C07278=1030.289,161.461,393.307,169.169,44.738,158.424
C07279=1030.283,161.212,393.329,169.167,44.740,158.424
C07280=1030.277,160.963,393.352,169.164,44.742,158.424
C07281=1030.272,160.714,393.374,169.160,44.744,158.424
C07282=1030.266,160.465,393.396,169.158,44.746,158.425
C07283=1030.260,160.216,393.419,169.155,44.748,158.425
C07284=1030.255,159.967,393.442,169.152,44.749,158.425
C07285=1030.249,159.718,393.464,169.149,44.751,158.425
C07286=1030.243,159.469,393.486,169.145,44.754,158.425
C07287=1030.237,159.220,393.508,169.143,44.756,158.425
C07288=1030.231,158.971,393.531,169.141,44.758,158.425
C07289=1030.225,158.722,393.552,169.137,44.760,158.425
C07290=1030.218,158.473,393.575,169.134,44.762,158.425
C07291=1030.213,158.224,393.597,169.131,44.764,158.426
C07292=1030.207,157.975,393.618,169.128,44.766,158.426
C07293=1030.201,157.727,393.641,169.126,44.769,158.426
C07294=1030.195,157.477,393.663,169.122,44.771,158.426
C07295=1030.189,157.229,393.685,169.120,44.773,158.426
C07296=1030.183,156.980,393.707,169.116,44.775,158.426
C07297=1030.176,156.695,393.733,169.113,44.777,158.426
C07298=1030.170,156.411,393.757,169.110,44.780,158.427
C07299=1030.162,156.127,393.782,169.107,44.782,158.427
C07300=1030.156,155.842,393.807,169.103,44.785,158.427
C07301=1030.149,155.593,393.830,169.100,44.787,158.427
C07302=1030.144,155.344,393.851,169.097,44.789,158.427
C07303=1030.138,155.095,393.873,169.095,44.791,158.427
C07304=1030.132,154.846,393.895,169.091,44.794,158.428
C07305=1030.126,154.597,393.917,169.089,44.796,158.428
C07306=1030.120,154.348,393.939,169.086,44.798,158.428
C07307=1030.115,154.099,393.961,169.083,44.800,158.428
C07308=1030.108,153.851,393.983,169.080,44.802,158.428
C07309=1030.102,153.601,394.005,169.078,44.804,158.428
C07310=1030.096,153.352,394.026,169.074,44.807,158.429
C07311=1030.091,153.103,394.048,169.072,44.808,158.429
C07312=1030.085,152.855,394.070,169.068,44.811,158.429
C07313=1030.078,152.606,394.092,169.066,44.813,158.429
C07314=1030.072,152.356,394.114,169.063,44.815,158.429
C07315=1030.066,152.107,394.135,169.060,44.817,158.429
C07316=1030.060,151.859,394.157,169.057,44.819,158.429
C07317=1030.054,151.609,394.178,169.055,44.821,158.430
C07318=1030.049,151.360,394.201,169.051,44.823,158.430
C07319=1030.042,151.111,394.223,169.049,44.826,158.430
C07320=1030.037,150.863,394.244,169.046,44.828,158.430
C07321=1030.031,150.614,394.266,169.043,44.830,158.430
C07322=1030.025,150.364,394.287,169.040,44.832,158.430
C07323=1030.018,150.115,394.309,169.038,44.835,158.431
C07324=1030.013,149.867,394.330,169.034,44.837,158.431
C07325=1030.007,149.617,394.352,169.032,44.839,158.431
C07326=1030.000,149.368,394.373,169.029,44.841,158.431
C07327=1029.996,149.119,394.395,169.026,44.844,158.431
C07328=1029.989,148.870,394.417,169.023,44.846,158.431
C07329=1029.983,148.621,394.439,169.021,44.848,158.431
C07330=1029.977,148.373,394.461,169.017,44.850,158.431
C07331=1029.971,148.124,394.482,169.015,44.852,158.432
C07332=1029.965,147.875,394.504,169.012,44.854,158.432
C07333=1029.959,147.626,394.525,169.009,44.856,158.432
C07334=1029.953,147.377,394.547,169.006,44.858,158.432
C07335=1029.948,147.127,394.568,169.004,44.861,158.432
C07336=1029.941,146.878,394.589,169.000,44.863,158.433
C07337=1029.936,146.629,394.611,168.998,44.865,158.433
C07338=1029.930,146.380,394.632,168.995,44.867,158.433
C07339=1029.924,146.131,394.654,168.992,44.870,158.433
C07340=1029.918,145.883,394.675,168.989,44.872,158.433
C07341=1029.912,145.633,394.697,168.987,44.874,158.433
C07342=1029.905,145.384,394.718,168.983,44.877,158.434
C07343=1029.899,145.136,394.739,168.981,44.879,158.434
C07344=1029.893,144.887,394.761,168.978,44.881,158.434
C07345=1029.887,144.637,394.782,168.975,44.883,158.434
C07346=1029.882,144.388,394.803,168.972,44.885,158.434
C07347=1029.876,144.139,394.825,168.970,44.888,158.434
C07348=1029.869,143.890,394.846,168.967,44.890,158.435
C07349=1029.863,143.642,394.867,168.964,44.892,158.435
C07350=1029.857,143.392,394.888,168.962,44.895,158.435
C07351=1029.852,143.143,394.909,168.959,44.897,158.435
C07352=1029.846,142.894,394.931,168.955,44.899,158.435
C07353=1029.839,142.645,394.952,168.953,44.901,158.435
C07354=1029.834,142.397,394.974,168.951,44.903,158.436
C07355=1029.828,142.147,394.994,168.947,44.906,158.436
C07356=1029.822,141.899,395.015,168.945,44.908,158.436
C07357=1029.815,141.649,395.037,168.942,44.910,158.436
C07358=1029.809,141.400,395.058,168.940,44.912,158.436
C07359=1029.804,141.151,395.079,168.936,44.915,158.436
C07360=1029.798,140.902,395.101,168.934,44.917,158.437
C07361=1029.791,140.618,395.125,168.930,44.920,158.437
C07362=1029.784,140.333,395.149,168.928,44.922,158.437
C07363=1029.778,140.047,395.173,168.924,44.925,158.437
C07364=1029.771,139.763,395.197,168.921,44.927,158.437
C07365=1029.765,139.514,395.219,168.919,44.929,158.438
C07366=1029.759,139.265,395.239,168.916,44.931,158.438
C07367=1029.753,139.016,395.260,168.913,44.934,158.438
C07368=1029.747,138.768,395.282,168.910,44.936,158.438
C07369=1029.741,138.518,395.303,168.908,44.938,158.438
C07370=1029.735,138.269,395.323,168.905,44.941,158.438
C07371=1029.729,138.020,395.344,168.902,44.943,158.439
C07372=1029.723,137.770,395.366,168.899,44.946,158.439
C07373=1029.717,137.522,395.387,168.897,44.947,158.439
C07374=1029.711,137.272,395.407,168.893,44.950,158.439
C07375=1029.705,137.024,395.429,168.891,44.952,158.439
C07376=1029.699,136.774,395.449,168.888,44.954,158.439
C07377=1029.693,136.526,395.470,168.886,44.957,158.440
C07378=1029.687,136.276,395.491,168.883,44.959,158.440
C07379=1029.681,136.028,395.512,168.880,44.962,158.440
C07380=1029.675,135.778,395.533,168.878,44.964,158.440
C07381=1029.669,135.530,395.554,168.875,44.966,158.440
C07382=1029.663,135.280,395.574,168.872,44.968,158.441
C07383=1029.657,135.032,395.596,168.869,44.970,158.441
C07384=1029.651,134.782,395.616,168.867,44.973,158.441
C07385=1029.645,134.534,395.637,168.864,44.975,158.441
C07386=1029.638,134.284,395.658,168.861,44.978,158.441
C07387=1029.633,134.035,395.678,168.859,44.980,158.442
C07388=1029.627,133.786,395.700,168.856,44.982,158.442
C07389=1029.621,133.537,395.720,168.854,44.984,158.442
C07390=1029.615,133.288,395.741,168.850,44.987,158.442
C07391=1029.609,133.039,395.761,168.848,44.989,158.442
C07392=1029.603,132.789,395.782,168.845,44.991,158.442
C07393=1029.597,132.541,395.803,168.843,44.994,158.443
C07394=1029.591,132.292,395.824,168.839,44.996,158.443
C07395=1029.585,132.043,395.845,168.837,44.999,158.443
C07396=1029.579,131.794,395.865,168.834,45.001,158.443
C07397=1029.573,131.544,395.886,168.832,45.003,158.443
C07398=1029.567,131.296,395.907,168.830,45.005,158.444
C07399=1029.561,131.046,395.928,168.826,45.007,158.444
C07400=1029.555,130.797,395.948,168.824,45.010,158.444
C07401=1029.550,130.549,395.969,168.821,45.012,158.444
C07402=1029.543,130.299,395.989,168.819,45.015,158.444
C07403=1029.538,130.050,396.010,168.815,45.017,158.445
C07404=1029.531,129.800,396.030,168.813,45.019,158.445
C07405=1029.525,129.552,396.050,168.810,45.021,158.445
C07406=1029.518,129.303,396.071,168.808,45.024,158.445
C07407=1029.513,129.054,396.092,168.805,45.027,158.445
C07408=1029.507,128.804,396.112,168.802,45.029,158.446
C07409=1029.501,128.555,396.132,168.800,45.032,158.446
C07410=1029.494,128.306,396.152,168.797,45.033,158.446
C07411=1029.488,128.057,396.172,168.794,45.036,158.446
C07412=1029.482,127.808,396.193,168.792,45.038,158.446
C07413=1029.476,127.559,396.214,168.789,45.041,158.447
C07414=1029.470,127.310,396.234,168.787,45.044,158.447
C07415=1029.463,127.061,396.254,168.783,45.046,158.447
C07416=1029.458,126.811,396.275,168.781,45.048,158.447
C07417=1029.452,126.563,396.295,168.779,45.050,158.447
C07418=1029.445,126.313,396.315,168.776,45.053,158.448
C07419=1029.439,126.064,396.335,168.773,45.056,158.448
C07420=1029.434,125.814,396.356,168.770,45.058,158.448
C07421=1029.427,125.566,396.376,168.768,45.060,158.448
C07422=1029.421,125.317,396.396,168.766,45.062,158.448
C07423=1029.415,125.068,396.417,168.763,45.065,158.449
C07424=1029.409,124.819,396.437,168.760,45.067,158.449
C07425=1029.403,124.575,396.457,168.757,45.070,158.449
C07426=1029.397,124.332,396.476,168.755,45.072,158.449
C07427=1029.391,124.088,396.496,168.752,45.075,158.450
C07428=1029.386,123.845,396.516,168.750,45.077,158.450
C07429=1029.380,123.602,396.536,168.748,45.079,158.450
C07430=1029.374,123.358,396.555,168.744,45.081,158.450
C07431=1029.368,123.115,396.575,168.742,45.084,158.450
C07432=1029.362,122.871,396.595,168.739,45.086,158.450
C07433=1029.356,122.622,396.615,168.737,45.089,158.451
C07434=1029.350,122.373,396.635,168.734,45.091,158.451
C07435=1029.344,122.124,396.655,168.732,45.093,158.451
C07436=1029.337,121.875,396.675,168.728,45.095,158.451
C07437=1029.332,121.625,396.696,168.726,45.098,158.451
C07438=1029.326,121.377,396.716,168.724,45.101,158.452
C07439=1029.320,121.127,396.736,168.721,45.103,158.452
C07440=1029.314,120.878,396.756,168.719,45.105,158.452
C07441=1029.308,120.629,396.777,168.716,45.107,158.452
C07442=1029.302,120.380,396.797,168.713,45.110,158.453
C07443=1029.296,120.131,396.817,168.711,45.112,158.453
C07444=1029.290,119.882,396.837,168.708,45.115,158.453
C07445=1029.284,119.633,396.856,168.706,45.117,158.453
C07446=1029.279,119.383,396.877,168.703,45.119,158.453
C07447=1029.272,119.134,396.897,168.701,45.121,158.454
C07448=1029.266,118.885,396.917,168.698,45.124,158.454
C07449=1029.260,118.636,396.937,168.695,45.126,158.454
C07450=1029.254,118.388,396.957,168.693,45.129,158.454
C07451=1029.248,118.138,396.978,168.690,45.131,158.454
C07452=1029.242,117.889,396.998,168.688,45.134,158.455
C07453=1029.235,117.592,397.021,168.685,45.136,158.455
C07454=1029.229,117.296,397.045,168.681,45.139,158.455
C07455=1029.221,117.001,397.069,168.679,45.142,158.455
C07456=1029.214,116.704,397.093,168.676,45.145,158.456
C07457=1029.208,116.455,397.113,168.673,45.147,158.456
C07458=1029.202,116.206,397.133,168.671,45.149,158.456
C07459=1029.197,115.957,397.152,168.668,45.151,158.456
C07460=1029.190,115.707,397.172,168.665,45.154,158.456
C07461=1029.185,115.458,397.193,168.662,45.156,158.456
C07462=1029.179,115.209,397.213,168.660,45.159,158.457
C07463=1029.173,114.960,397.232,168.658,45.161,158.457
C07464=1029.167,114.711,397.252,168.655,45.164,158.457
C07465=1029.161,114.462,397.272,168.653,45.165,158.457
C07466=1029.155,114.213,397.292,168.650,45.167,158.457
C07467=1029.150,113.963,397.312,168.648,45.170,158.458
C07468=1029.144,113.714,397.332,168.644,45.172,158.458
C07469=1029.138,113.465,397.352,168.642,45.175,158.458
C07470=1029.132,113.217,397.372,168.639,45.177,158.458
C07471=1029.126,112.967,397.391,168.637,45.180,158.458
C07472=1029.119,112.718,397.412,168.635,45.182,158.459
C07473=1029.114,112.468,397.431,168.632,45.184,158.459
C07474=1029.108,112.219,397.451,168.630,45.187,158.459
C07475=1029.102,111.971,397.471,168.627,45.189,158.459
C07476=1029.096,111.721,397.490,168.624,45.192,158.459
C07477=1029.090,111.472,397.510,168.622,45.194,158.460
C07478=1029.084,111.222,397.530,168.619,45.196,158.460
C07479=1029.078,110.973,397.550,168.617,45.199,158.460
C07480=1029.072,110.724,397.569,168.614,45.201,158.460
C07481=1029.065,110.475,397.588,168.612,45.204,158.461
C07482=1029.059,110.227,397.608,168.610,45.206,158.461
C07483=1029.054,109.977,397.627,168.606,45.209,158.461
C07484=1029.048,109.728,397.647,168.604,45.211,158.461
C07485=1029.041,109.478,397.667,168.601,45.213,158.461
C07486=1029.035,109.229,397.686,168.599,45.216,158.462
C07487=1029.029,108.980,397.706,168.597,45.219,158.462
C07488=1029.023,108.731,397.725,168.594,45.220,158.462
C07489=1029.016,108.447,397.747,168.591,45.223,158.462
C07490=1029.009,108.162,397.769,168.588,45.227,158.463
C07491=1029.002,107.877,397.791,168.586,45.230,158.463
C07492=1028.995,107.591,397.814,168.582,45.232,158.463
C07493=1028.989,107.342,397.834,168.580,45.234,158.463
C07494=1028.983,107.093,397.853,168.577,45.237,158.463
C07495=1028.977,106.844,397.872,168.575,45.240,158.464
C07496=1028.971,106.595,397.892,168.573,45.242,158.464
C07497=1028.965,106.345,397.911,168.569,45.245,158.464
C07498=1028.959,106.096,397.929,168.567,45.247,158.464
C07499=1028.953,105.847,397.949,168.564,45.249,158.464
C07500=1028.947,105.598,397.969,168.562,45.252,158.465
C07501=1028.941,105.349,397.989,168.560,45.254,158.465
C07502=1028.935,105.100,398.007,168.557,45.257,158.465
C07503=1028.929,104.851,398.027,168.555,45.259,158.465
C07504=1028.922,104.601,398.047,168.553,45.261,158.466
C07505=1028.916,104.352,398.065,168.549,45.264,158.466
C07506=1028.910,104.102,398.085,168.547,45.267,158.466
C07507=1028.905,103.853,398.104,168.544,45.269,158.466
C07508=1028.899,103.604,398.124,168.542,45.271,158.466
C07509=1028.892,103.355,398.143,168.540,45.273,158.467
C07510=1028.886,103.106,398.162,168.537,45.276,158.467
C07511=1028.880,102.857,398.182,168.535,45.279,158.467
C07512=1028.874,102.608,398.200,168.532,45.281,158.467
C07513=1028.868,102.358,398.220,168.530,45.283,158.468
C07514=1028.863,102.109,398.239,168.527,45.286,158.468
C07515=1028.857,101.860,398.259,168.524,45.288,158.468
C07516=1028.850,101.611,398.278,168.522,45.291,158.468
C07517=1028.845,101.362,398.297,168.519,45.293,158.468
C07518=1028.839,101.112,398.316,168.517,45.296,158.469
C07519=1028.832,100.864,398.335,168.515,45.298,158.469
C07520=1028.826,100.614,398.355,168.512,45.300,158.469
C07521=1028.821,100.365,398.374,168.510,45.303,158.469
C07522=1028.815,100.115,398.393,168.507,45.305,158.469
C07523=1028.809,99.866,398.412,168.505,45.308,158.470
C07524=1028.803,99.617,398.431,168.502,45.310,158.470
C07525=1028.796,99.368,398.450,168.499,45.312,158.470
C07526=1028.791,99.119,398.470,168.497,45.315,158.470
C07527=1028.784,98.870,398.488,168.495,45.318,158.471
C07528=1028.778,98.621,398.507,168.492,45.320,158.471
C07529=1028.772,98.371,398.526,168.490,45.322,158.471
C07530=1028.766,98.122,398.545,168.488,45.325,158.471
C07531=1028.760,97.873,398.564,168.484,45.328,158.471
C07532=1028.753,97.623,398.583,168.482,45.330,158.472
C07533=1028.748,97.374,398.602,168.479,45.333,158.472
C07534=1028.741,97.125,398.621,168.477,45.335,158.472
C07535=1028.735,96.876,398.639,168.475,45.337,158.472
C07536=1028.729,96.626,398.658,168.472,45.340,158.473
C07537=1028.723,96.378,398.677,168.470,45.343,158.473
C07538=1028.718,96.128,398.696,168.468,45.345,158.473
C07539=1028.711,95.879,398.715,168.464,45.348,158.473
C07540=1028.705,95.630,398.733,168.462,45.350,158.473
C07541=1028.699,95.381,398.753,168.460,45.353,158.474
C07542=1028.693,95.132,398.771,168.457,45.355,158.474
C07543=1028.687,94.882,398.790,168.455,45.358,158.474
C07544=1028.681,94.633,398.809,168.452,45.360,158.474
C07545=1028.675,94.384,398.828,168.450,45.362,158.474
C07546=1028.669,94.135,398.847,168.448,45.365,158.475
C07547=1028.662,93.885,398.866,168.445,45.368,158.475
C07548=1028.656,93.636,398.885,168.443,45.370,158.475
C07549=1028.651,93.388,398.903,168.439,45.373,158.475
C07550=1028.645,93.138,398.922,168.437,45.375,158.476
C07551=1028.638,92.889,398.941,168.435,45.377,158.476
C07552=1028.632,92.639,398.959,168.432,45.380,158.476
C07553=1028.626,92.354,398.981,168.430,45.383,158.476
C07554=1028.619,92.069,399.003,168.427,45.385,158.477
C07555=1028.611,91.784,399.024,168.424,45.388,158.477
C07556=1028.605,91.500,399.045,168.421,45.391,158.477
C07557=1028.599,91.251,399.064,168.419,45.394,158.477
C07558=1028.593,91.001,399.083,168.416,45.396,158.477
C07559=1028.587,90.752,399.102,168.414,45.398,158.478
C07560=1028.581,90.502,399.120,168.412,45.401,158.478
C07561=1028.575,90.253,399.139,168.409,45.403,158.478
C07562=1028.568,90.004,399.158,168.407,45.406,158.478
C07563=1028.563,89.755,399.176,168.405,45.408,158.479
C07564=1028.557,89.506,399.195,168.401,45.411,158.479
C07565=1028.551,89.256,399.213,168.399,45.413,158.479
C07566=1028.544,89.007,399.232,168.397,45.416,158.479
C07567=1028.538,88.758,399.250,168.394,45.419,158.480
C07568=1028.533,88.508,399.269,168.392,45.421,158.480
C07569=1028.526,88.259,399.288,168.389,45.423,158.480
C07570=1028.520,88.010,399.306,168.387,45.426,158.480
C07571=1028.514,87.761,399.324,168.385,45.429,158.480
C07572=1028.508,87.511,399.342,168.381,45.431,158.481
C07573=1028.501,87.262,399.361,168.379,45.434,158.481
C07574=1028.495,87.013,399.379,168.377,45.436,158.481
C07575=1028.489,86.763,399.398,168.374,45.439,158.481
C07576=1028.483,86.515,399.416,168.372,45.442,158.482
C07577=1028.478,86.265,399.434,168.370,45.444,158.482
C07578=1028.471,86.016,399.453,168.367,45.446,158.482
C07579=1028.465,85.767,399.472,168.365,45.449,158.482
C07580=1028.459,85.517,399.490,168.363,45.452,158.483
C07581=1028.453,85.269,399.508,168.359,45.454,158.483
C07582=1028.446,85.019,399.527,168.357,45.457,158.483
C07583=1028.440,84.770,399.545,168.355,45.459,158.483
C07584=1028.434,84.521,399.563,168.352,45.461,158.483
C07585=1028.428,84.271,399.581,168.350,45.464,158.484
C07586=1028.422,84.022,399.599,168.347,45.467,158.484
C07587=1028.416,83.773,399.617,168.345,45.469,158.484
C07588=1028.410,83.523,399.637,168.343,45.471,158.484
C07589=1028.404,83.274,399.655,168.340,45.474,158.484
C07590=1028.398,83.025,399.673,168.338,45.477,158.485
C07591=1028.392,82.776,399.691,168.335,45.479,158.485
C07592=1028.386,82.526,399.709,168.332,45.482,158.485
C07593=1028.379,82.277,399.728,168.330,45.484,158.485
C07594=1028.374,82.028,399.746,168.328,45.487,158.486
C07595=1028.367,81.779,399.764,168.325,45.489,158.486
C07596=1028.361,81.529,399.782,168.323,45.492,158.486
C07597=1028.355,81.280,399.801,168.321,45.494,158.486
C07598=1028.349,81.031,399.818,168.318,45.496,158.486
C07599=1028.343,80.782,399.837,168.316,45.499,158.487
C07600=1028.337,80.532,399.856,168.313,45.502,158.487
C07601=1028.331,80.283,399.874,168.311,45.504,158.487
C07602=1028.325,80.034,399.892,168.309,45.506,158.487
C07603=1028.319,79.785,399.910,168.306,45.509,158.488
C07604=1028.313,79.535,399.928,168.303,45.511,158.488
C07605=1028.307,79.286,399.947,168.301,45.514,158.488
C07606=1028.301,79.037,399.965,168.298,45.517,158.488
C07607=1028.295,78.787,399.982,168.296,45.519,158.488
C07608=1028.289,78.539,400.001,168.293,45.521,158.489
C07609=1028.283,78.289,400.019,168.291,45.524,158.489
C07610=1028.276,78.040,400.037,168.289,45.526,158.489
C07611=1028.271,77.791,400.055,168.286,45.529,158.489
C07612=1028.265,77.541,400.073,168.284,45.532,158.490
C07613=1028.258,77.292,400.091,168.281,45.534,158.490
C07614=1028.253,77.043,400.109,168.279,45.536,158.490
C07615=1028.247,76.793,400.127,168.277,45.539,158.490
C07616=1028.240,76.544,400.146,168.275,45.542,158.490
C07617=1028.234,76.259,400.166,168.271,45.545,158.491
C07618=1028.226,75.974,400.187,168.268,45.547,158.491
C07619=1028.219,75.689,400.207,168.266,45.550,158.491
C07620=1028.213,75.403,400.227,168.262,45.553,158.491
C07621=1028.206,75.154,400.246,168.260,45.556,158.492
C07622=1028.199,74.905,400.263,168.258,45.558,158.492
C07623=1028.194,74.656,400.280,168.256,45.561,158.492
C07624=1028.188,74.406,400.298,168.253,45.563,158.492
C07625=1028.182,74.158,400.317,168.251,45.566,158.493
C07626=1028.176,73.908,400.335,168.249,45.569,158.493
C07627=1028.169,73.659,400.352,168.246,45.571,158.493
C07628=1028.163,73.409,400.369,168.244,45.573,158.493
C07629=1028.157,73.160,400.387,168.240,45.576,158.493
C07630=1028.151,72.911,400.406,168.238,45.579,158.494
C07631=1028.145,72.662,400.424,168.236,45.581,158.494
C07632=1028.139,72.412,400.441,168.233,45.584,158.494
C07633=1028.133,72.163,400.459,168.231,45.586,158.494
C07634=1028.127,71.913,400.476,168.229,45.589,158.495
C07635=1028.120,71.664,400.495,168.226,45.591,158.495
C07636=1028.115,71.415,400.513,168.224,45.594,158.495
C07637=1028.108,71.166,400.530,168.222,45.596,158.495
C07638=1028.103,70.917,400.548,168.219,45.599,158.496
C07639=1028.096,70.667,400.566,168.217,45.601,158.496
C07640=1028.090,70.418,400.583,168.215,45.604,158.496
C07641=1028.084,70.169,400.600,168.211,45.607,158.496
C07642=1028.078,69.919,400.618,168.209,45.609,158.496
C07643=1028.072,69.670,400.636,168.206,45.611,158.496
C07644=1028.065,69.421,400.654,168.204,45.614,158.497
C07645=1028.060,69.172,400.672,168.202,45.617,158.497
C07646=1028.054,68.922,400.689,168.199,45.619,158.497
C07647=1028.047,68.672,400.707,168.197,45.622,158.497
C07648=1028.041,68.424,400.724,168.195,45.624,158.498
C07649=1028.035,68.174,400.742,168.193,45.627,158.498
C07650=1028.029,67.925,400.759,168.190,45.629,158.498
C07651=1028.023,67.675,400.777,168.188,45.632,158.498
C07652=1028.017,67.426,400.795,168.184,45.635,158.499
C07653=1028.010,67.177,400.812,168.182,45.637,158.499
C07654=1028.005,66.928,400.830,168.180,45.639,158.499
C07655=1027.999,66.678,400.848,168.177,45.642,158.499
C07656=1027.992,66.429,400.865,168.175,45.645,158.499
C07657=1027.986,66.180,400.883,168.173,45.647,158.500
C07658=1027.979,65.930,400.900,168.170,45.649,158.500
C07659=1027.974,65.681,400.917,168.168,45.652,158.500
C07660=1027.967,65.431,400.934,168.166,45.655,158.500
C07661=1027.962,65.182,400.952,168.163,45.658,158.501
C07662=1027.955,64.933,400.969,168.160,45.660,158.501
C07663=1027.950,64.684,400.987,168.158,45.663,158.501
C07664=1027.943,64.434,401.004,168.155,45.665,158.501
C07665=1027.937,64.185,401.021,168.153,45.668,158.501
C07666=1027.931,63.935,401.039,168.150,45.670,158.502
C07667=1027.925,63.687,401.056,168.148,45.673,158.502
C07668=1027.919,63.437,401.074,168.146,45.675,158.502
C07669=1027.913,63.188,401.091,168.144,45.678,158.502
C07670=1027.906,62.938,401.108,168.141,45.681,158.503
C07671=1027.900,62.689,401.125,168.138,45.684,158.503
C07672=1027.893,62.440,401.143,168.136,45.686,158.503
C07673=1027.887,62.190,401.159,168.133,45.688,158.503
C07674=1027.881,61.941,401.176,168.131,45.691,158.504
C07675=1027.875,61.692,401.194,168.129,45.694,158.504
C07676=1027.869,61.442,401.211,168.126,45.697,158.504
C07677=1027.862,61.193,401.228,168.124,45.699,158.504
C07678=1027.856,60.943,401.245,168.121,45.702,158.505
C07679=1027.850,60.695,401.262,168.119,45.705,158.505
C07680=1027.843,60.445,401.279,168.116,45.708,158.505
C07681=1027.836,60.160,401.298,168.113,45.711,158.505
C07682=1027.829,59.874,401.319,168.111,45.713,158.506
C07683=1027.822,59.590,401.338,168.107,45.716,158.506
C07684=1027.816,59.304,401.357,168.105,45.720,158.506
C07685=1027.809,59.055,401.375,168.103,45.722,158.506
C07686=1027.803,58.806,401.391,168.100,45.725,158.506
C07687=1027.796,58.556,401.408,168.097,45.727,158.507
C07688=1027.790,58.307,401.426,168.095,45.730,158.507
C07689=1027.784,58.057,401.442,168.093,45.733,158.507
C07690=1027.778,57.808,401.459,168.091,45.735,158.508
C07691=1027.772,57.559,401.476,168.088,45.738,158.508
C07692=1027.765,57.309,401.494,168.086,45.740,158.508
C07693=1027.759,57.060,401.511,168.082,45.743,158.508
C07694=1027.753,56.810,401.527,168.080,45.746,158.508
C07695=1027.746,56.562,401.544,168.078,45.748,158.509
C07696=1027.740,56.312,401.561,168.076,45.751,158.509
C07697=1027.734,56.063,401.578,168.073,45.754,158.509
C07698=1027.728,55.814,401.595,168.071,45.756,158.509
C07699=1027.722,55.564,401.612,168.069,45.759,158.510
C07700=1027.715,55.315,401.629,168.066,45.761,158.510
C07701=1027.710,55.065,401.646,168.063,45.764,158.510
C07702=1027.703,54.816,401.663,168.061,45.767,158.510
C07703=1027.697,54.567,401.679,168.058,45.769,158.510
C07704=1027.690,54.317,401.697,168.056,45.772,158.511
C07705=1027.685,54.068,401.714,168.054,45.774,158.511
C07706=1027.679,53.819,401.730,168.051,45.777,158.511
C07707=1027.672,53.569,401.747,168.049,45.780,158.511
C07708=1027.666,53.320,401.764,168.047,45.782,158.512
C07709=1027.661,53.070,401.781,168.043,45.785,158.512
C07710=1027.654,52.821,401.798,168.041,45.788,158.512
C07711=1027.648,52.572,401.815,168.039,45.790,158.512
C07712=1027.642,52.323,401.832,168.036,45.792,158.512
C07713=1027.635,52.073,401.848,168.034,45.795,158.513
C07714=1027.630,51.824,401.866,168.032,45.798,158.513
C07715=1027.624,51.574,401.882,168.029,45.801,158.513
C07716=1027.617,51.325,401.899,168.027,45.803,158.513
C07717=1027.611,51.076,401.916,168.025,45.805,158.514
C07718=1027.605,50.827,401.933,168.021,45.808,158.514
C07719=1027.599,50.577,401.950,168.019,45.811,158.514
C07720=1027.593,50.327,401.966,168.016,45.813,158.514
C07721=1027.587,50.079,401.983,168.014,45.816,158.514
C07722=1027.581,49.829,401.999,168.012,45.818,158.515
C07723=1027.575,49.579,402.017,168.009,45.820,158.515
C07724=1027.569,49.330,402.033,168.007,45.823,158.515
C07725=1027.563,49.081,402.050,168.005,45.826,158.515
C07726=1027.556,48.832,402.067,168.003,45.829,158.516
C07727=1027.550,48.582,402.083,168.000,45.831,158.516
C07728=1027.544,48.333,402.101,167.997,45.834,158.516
C07729=1027.538,48.084,402.117,167.994,45.836,158.516
C07730=1027.532,47.834,402.134,167.992,45.838,158.516
C07731=1027.526,47.585,402.151,167.990,45.841,158.516
C07732=1027.520,47.335,402.167,167.987,45.844,158.517
C07733=1027.514,47.086,402.184,167.985,45.846,158.517
C07734=1027.508,46.837,402.201,167.983,45.849,158.517
C07735=1027.502,46.587,402.217,167.980,45.851,158.517
C07736=1027.496,46.338,402.234,167.978,45.853,158.517
C07737=1027.489,46.089,402.251,167.976,45.856,158.518
C07738=1027.484,45.839,402.267,167.973,45.859,158.518
C07739=1027.478,45.589,402.284,167.971,45.861,158.518
C07740=1027.472,45.340,402.300,167.967,45.864,158.518
C07741=1027.466,45.091,402.317,167.965,45.866,158.519
C07742=1027.460,44.842,402.334,167.963,45.869,158.519
C07743=1027.454,44.592,402.350,167.960,45.871,158.519
C07744=1027.448,44.343,402.367,167.958,45.873,158.519
C07745=1027.441,44.057,402.386,167.956,45.876,158.519
C07746=1027.434,43.772,402.406,167.952,45.879,158.519
C07747=1027.428,43.486,402.424,167.950,45.882,158.520
C07748=1027.420,43.201,402.443,167.947,45.885,158.520
C07749=1027.415,42.951,402.460,167.944,45.887,158.520
C07750=1027.409,42.702,402.476,167.942,45.890,158.520
C07751=1027.403,42.452,402.493,167.940,45.893,158.521
C07752=1027.396,42.203,402.508,167.937,45.895,158.521
C07753=1027.389,41.953,402.525,167.934,45.898,158.521
C07754=1027.383,41.705,402.542,167.932,45.901,158.521
C07755=1027.377,41.455,402.558,167.930,45.903,158.522
C07756=1027.371,41.206,402.574,167.927,45.905,158.522
C07757=1027.365,40.957,402.591,167.925,45.908,158.522
C07758=1027.359,40.707,402.607,167.923,45.911,158.522
C07759=1027.353,40.457,402.624,167.920,45.914,158.522
C07760=1027.347,40.208,402.640,167.918,45.916,158.523
C07761=1027.341,39.958,402.656,167.914,45.919,158.523
C07762=1027.335,39.709,402.672,167.912,45.921,158.523
C07763=1027.328,39.460,402.688,167.910,45.924,158.523
C07764=1027.322,39.211,402.704,167.907,45.926,158.523
C07765=1027.316,38.961,402.720,167.905,45.929,158.524
C07766=1027.310,38.711,402.737,167.903,45.931,158.524
C07767=1027.304,38.462,402.753,167.901,45.934,158.524
C07768=1027.298,38.213,402.770,167.898,45.936,158.524
C07769=1027.292,37.963,402.786,167.895,45.939,158.524
C07770=1027.286,37.714,402.802,167.893,45.942,158.525
C07771=1027.280,37.465,402.818,167.890,45.944,158.525
C07772=1027.274,37.215,402.835,167.888,45.947,158.525
C07773=1027.268,36.966,402.851,167.885,45.949,158.525
C07774=1027.261,36.716,402.867,167.883,45.952,158.526
C07775=1027.255,36.467,402.883,167.881,45.954,158.526
C07776=1027.249,36.217,402.899,167.877,45.957,158.526
C07777=1027.242,35.968,402.915,167.875,45.960,158.526
C07778=1027.237,35.718,402.931,167.873,45.963,158.526
C07779=1027.231,35.469,402.947,167.871,45.965,158.527
C07780=1027.224,35.220,402.963,167.868,45.968,158.527
C07781=1027.218,34.971,402.979,167.865,45.970,158.527
C07782=1027.212,34.721,402.995,167.862,45.973,158.527
C07783=1027.205,34.472,403.011,167.860,45.976,158.527
C07784=1027.200,34.222,403.026,167.858,45.979,158.528
C07785=1027.193,33.972,403.043,167.856,45.981,158.528
C07786=1027.187,33.723,403.059,167.853,45.983,158.528
C07787=1027.181,33.474,403.075,167.850,45.986,158.528
C07788=1027.175,33.225,403.091,167.848,45.989,158.528
C07789=1027.168,32.975,403.106,167.845,45.992,158.529
C07790=1027.162,32.726,403.122,167.843,45.995,158.529
C07791=1027.156,32.476,403.139,167.841,45.997,158.529
C07792=1027.150,32.227,403.154,167.838,45.999,158.529
C07793=1027.144,31.978,403.170,167.835,46.002,158.530
C07794=1027.138,31.728,403.186,167.833,46.005,158.530
C07795=1027.131,31.479,403.202,167.830,46.007,158.530
C07796=1027.125,31.230,403.218,167.828,46.010,158.530
C07797=1027.119,30.980,403.234,167.826,46.013,158.530
C07798=1027.113,30.730,403.249,167.823,46.015,158.531
C07799=1027.107,30.481,403.265,167.820,46.018,158.531
C07800=1027.100,30.232,403.281,167.818,46.020,158.531
C07801=1027.095,29.982,403.297,167.815,46.023,158.531
C07802=1027.089,29.733,403.313,167.813,46.026,158.531
C07803=1027.082,29.484,403.328,167.811,46.028,158.532
C07804=1027.077,29.234,403.344,167.808,46.031,158.532
C07805=1027.071,28.984,403.360,167.805,46.034,158.532
C07806=1027.064,28.735,403.376,167.803,46.036,158.532
C07807=1027.058,28.485,403.391,167.800,46.038,158.532
C07808=1027.052,28.236,403.408,167.798,46.041,158.533
C07809=1027.045,27.951,403.425,167.795,46.044,158.533
C07810=1027.038,27.665,403.444,167.792,46.047,158.533
C07811=1027.031,27.380,403.462,167.789,46.050,158.533
C07812=1027.024,27.094,403.479,167.786,46.054,158.534
C07813=1027.018,26.845,403.495,167.784,46.056,158.534
C07814=1027.011,26.596,403.511,167.781,46.058,158.534
C07815=1027.005,26.346,403.526,167.779,46.061,158.534
C07816=1026.999,26.097,403.542,167.777,46.064,158.534
C07817=1026.993,25.847,403.557,167.774,46.067,158.535
C07818=1026.987,25.598,403.573,167.771,46.069,158.535
C07819=1026.980,25.348,403.588,167.769,46.072,158.535
C07820=1026.974,25.099,403.604,167.767,46.074,158.535
C07821=1026.968,24.849,403.619,167.764,46.077,158.536
C07822=1026.961,24.600,403.635,167.761,46.080,158.536
C07823=1026.956,24.350,403.651,167.759,46.083,158.536
C07824=1026.949,24.101,403.666,167.756,46.085,158.536
C07825=1026.944,23.852,403.681,167.754,46.088,158.536
C07826=1026.937,23.602,403.696,167.752,46.090,158.537
C07827=1026.932,23.353,403.713,167.748,46.093,158.537
C07828=1026.925,23.103,403.728,167.746,46.096,158.537
C07829=1026.918,22.854,403.743,167.744,46.098,158.537
C07830=1026.913,22.604,403.759,167.741,46.101,158.537
C07831=1026.906,22.355,403.774,167.739,46.104,158.538
C07832=1026.900,22.105,403.790,167.736,46.107,158.538
C07833=1026.894,21.855,403.805,167.733,46.109,158.538
C07834=1026.888,21.607,403.820,167.731,46.111,158.538
C07835=1026.882,21.357,403.836,167.729,46.114,158.538
C07836=1026.876,21.108,403.851,167.727,46.117,158.539
C07837=1026.869,20.858,403.866,167.723,46.119,158.539
C07838=1026.864,20.608,403.882,167.721,46.122,158.539
C07839=1026.857,20.359,403.898,167.718,46.125,158.539
C07840=1026.851,20.109,403.913,167.716,46.128,158.539
C07841=1026.845,19.860,403.928,167.714,46.130,158.540
C07842=1026.839,19.611,403.943,167.710,46.133,158.540
C07843=1026.833,19.361,403.959,167.708,46.135,158.540
C07844=1026.827,19.112,403.974,167.706,46.138,158.540
C07845=1026.820,18.863,403.990,167.703,46.140,158.540
C07846=1026.814,18.613,404.005,167.700,46.143,158.541
C07847=1026.808,18.363,404.020,167.698,46.146,158.541
C07848=1026.802,18.114,404.035,167.696,46.149,158.541
C07849=1026.796,17.865,404.050,167.693,46.151,158.541
C07850=1026.790,17.615,404.066,167.691,46.153,158.541
C07851=1026.784,17.365,404.081,167.688,46.156,158.542
C07852=1026.777,17.116,404.096,167.685,46.159,158.542
C07853=1026.771,16.866,404.111,167.683,46.162,158.542
C07854=1026.765,16.618,404.126,167.681,46.165,158.542
C07855=1026.759,16.368,404.141,167.677,46.167,158.542
C07856=1026.753,16.118,404.156,167.675,46.170,158.543
C07857=1026.746,15.868,404.171,167.673,46.172,158.543
C07858=1026.740,15.619,404.186,167.670,46.175,158.543
C07859=1026.735,15.370,404.202,167.668,46.177,158.543
C07860=1026.728,15.121,404.217,167.665,46.180,158.543
C07861=1026.722,14.871,404.232,167.662,46.183,158.544
C07862=1026.715,14.621,404.247,167.660,46.186,158.544
C07863=1026.710,14.372,404.262,167.658,46.188,158.544
C07864=1026.704,14.122,404.277,167.654,46.191,158.544
C07865=1026.698,13.873,404.292,167.652,46.194,158.544
C07866=1026.691,13.624,404.308,167.650,46.196,158.545
C07867=1026.685,13.375,404.322,167.648,46.199,158.545
C07868=1026.679,13.125,404.337,167.644,46.201,158.545
C07869=1026.672,12.875,404.352,167.642,46.204,158.545
C07870=1026.666,12.626,404.367,167.640,46.207,158.545
C07871=1026.660,12.376,404.382,167.636,46.210,158.546
C07872=1026.654,12.127,404.397,167.634,46.213,158.546
C07873=1026.647,11.843,404.414,167.631,46.216,158.546
C07874=1026.639,11.558,404.431,167.629,46.219,158.546
C07875=1026.633,11.274,404.447,167.625,46.222,158.547
C07876=1026.626,10.990,404.464,167.622,46.225,158.547
C07877=1026.619,10.740,404.479,167.620,46.228,158.547
C07878=1026.613,10.490,404.494,167.618,46.231,158.547
C07879=1026.607,10.241,404.508,167.614,46.234,158.548
C07880=1026.601,9.992,404.523,167.612,46.236,158.548
C07881=1026.594,9.742,404.538,167.610,46.238,158.548
C07882=1026.588,9.493,404.553,167.606,46.241,158.548
C07883=1026.582,9.244,404.568,167.604,46.244,158.548
C07884=1026.576,8.994,404.583,167.602,46.247,158.549
C07885=1026.569,8.744,404.597,167.600,46.250,158.549
C07886=1026.563,8.495,404.612,167.596,46.253,158.549
C07887=1026.557,8.246,404.627,167.594,46.255,158.549
C07888=1026.550,7.996,404.641,167.592,46.258,158.549
C07889=1026.545,7.747,404.655,167.588,46.261,158.549
C07890=1026.538,7.497,404.670,167.586,46.263,158.550
C07891=1026.532,7.247,404.685,167.584,46.266,158.550
C07892=1026.526,6.998,404.700,167.582,46.269,158.550
C07893=1026.520,6.749,404.715,167.578,46.271,158.550
C07894=1026.513,6.498,404.729,167.576,46.274,158.551
C07895=1026.508,6.250,404.743,167.573,46.277,158.551
C07896=1026.501,6.000,404.758,167.570,46.280,158.551
C07897=1026.496,5.751,404.773,167.568,46.283,158.551
C07898=1026.489,5.501,404.788,167.565,46.285,158.551
C07899=1026.483,5.252,404.803,167.563,46.287,158.552
C07900=1026.477,5.002,404.817,167.560,46.290,158.552
C07901=1026.471,4.752,404.832,167.558,46.293,158.552
C07902=1026.465,4.503,404.847,167.555,46.295,158.552
C07903=1026.459,4.254,404.861,167.552,46.298,158.552
C07904=1026.452,4.004,404.875,167.550,46.301,158.552
C07905=1026.446,3.755,404.889,167.547,46.304,158.553
C07906=1026.440,3.505,404.904,167.545,46.307,158.553
C07907=1026.434,3.256,404.919,167.542,46.309,158.553
C07908=1026.428,3.006,404.933,167.539,46.312,158.553
C07909=1026.422,2.756,404.948,167.537,46.314,158.553
C07910=1026.416,2.507,404.963,167.534,46.317,158.554
C07911=1026.409,2.258,404.978,167.531,46.319,158.554
C07912=1026.404,2.008,404.991,167.529,46.322,158.554
C07913=1026.398,1.758,405.006,167.527,46.325,158.554
C07914=1026.392,1.510,405.021,167.523,46.327,158.554
C07915=1026.386,1.259,405.035,167.521,46.330,158.554
C07916=1026.379,1.010,405.050,167.519,46.333,158.555
C07917=1026.373,0.761,405.064,167.515,46.336,158.555
C07918=1026.367,0.511,405.078,167.513,46.338,158.555
C07919=1026.361,0.262,405.093,167.511,46.341,158.555
C07920=1026.355,0.012,405.108,167.508,46.343,158.556
C07921=1026.349,-0.238,405.122,167.505,46.346,158.556
C07922=1026.343,-0.487,405.137,167.503,46.349,158.556
C07923=1026.337,-0.736,405.151,167.500,46.351,158.556
C07924=1026.331,-0.986,405.166,167.497,46.354,158.556
C07925=1026.325,-1.235,405.180,167.495,46.356,158.556
C07926=1026.319,-1.486,405.194,167.492,46.359,158.557
C07927=1026.312,-1.734,405.208,167.490,46.362,158.557
C07928=1026.306,-1.984,405.223,167.487,46.364,158.557
C07929=1026.301,-2.234,405.237,167.484,46.367,158.557
C07930=1026.294,-2.483,405.252,167.482,46.370,158.557
C07931=1026.289,-2.733,405.266,167.480,46.372,158.557
C07932=1026.283,-2.982,405.281,167.476,46.375,158.558
C07933=1026.277,-3.232,405.295,167.474,46.378,158.558
C07934=1026.271,-3.481,405.309,167.471,46.380,158.558
C07935=1026.265,-3.731,405.324,167.468,46.383,158.558
C07936=1026.259,-3.980,405.338,167.466,46.386,158.558
C07937=1026.252,-4.263,405.354,167.463,46.389,158.558
C07938=1026.244,-4.544,405.370,167.460,46.391,158.559
C07939=1026.238,-4.827,405.386,167.457,46.394,158.559
C07940=1026.231,-5.110,405.401,167.454,46.398,158.559
C07941=1026.224,-5.359,405.416,167.452,46.400,158.559
C07942=1026.218,-5.609,405.429,167.448,46.403,158.559
C07943=1026.212,-5.859,405.443,167.446,46.406,158.560
C07944=1026.206,-6.108,405.457,167.443,46.409,158.560
C07945=1026.199,-6.358,405.472,167.441,46.412,158.560
C07946=1026.194,-6.607,405.486,167.438,46.415,158.560
C07947=1026.187,-6.857,405.500,167.435,46.418,158.561
C07948=1026.181,-7.106,405.514,167.433,46.420,158.561
C07949=1026.175,-7.356,405.527,167.430,46.422,158.561
C07950=1026.169,-7.605,405.542,167.427,46.425,158.561
C07951=1026.163,-7.854,405.555,167.425,46.428,158.561
C07952=1026.157,-8.105,405.570,167.422,46.431,158.561
C07953=1026.150,-8.353,405.583,167.419,46.434,158.562
C07954=1026.145,-8.603,405.597,167.417,46.436,158.562
C07955=1026.138,-8.853,405.611,167.414,46.439,158.562
C07956=1026.132,-9.103,405.625,167.411,46.442,158.562
C07957=1026.125,-9.352,405.639,167.409,46.445,158.562
C07958=1026.120,-9.601,405.653,167.406,46.448,158.563
C07959=1026.114,-9.851,405.667,167.403,46.450,158.563
C07960=1026.107,-10.101,405.681,167.401,46.453,158.563
C07961=1026.102,-10.350,405.695,167.398,46.456,158.563
C07962=1026.095,-10.599,405.708,167.396,46.458,158.563
C07963=1026.089,-10.849,405.723,167.392,46.461,158.563
C07964=1026.083,-11.099,405.736,167.390,46.464,158.564
C07965=1026.078,-11.348,405.750,167.387,46.466,158.564
C07966=1026.070,-11.598,405.764,167.384,46.469,158.564
C07967=1026.065,-11.847,405.778,167.382,46.472,158.564
C07968=1026.059,-12.096,405.791,167.379,46.474,158.564
C07969=1026.053,-12.347,405.806,167.376,46.477,158.565
C07970=1026.046,-12.596,405.819,167.374,46.480,158.565
C07971=1026.041,-12.846,405.833,167.372,46.483,158.565
C07972=1026.034,-13.095,405.847,167.368,46.485,158.565
C07973=1026.028,-13.345,405.861,167.366,46.488,158.565
C07974=1026.022,-13.594,405.874,167.363,46.491,158.565
C07975=1026.016,-13.844,405.888,167.360,46.494,158.566
C07976=1026.010,-14.093,405.902,167.358,46.496,158.566
C07977=1026.004,-14.343,405.915,167.355,46.499,158.566
C07978=1025.998,-14.592,405.929,167.352,46.502,158.566
C07979=1025.992,-14.842,405.943,167.350,46.504,158.566
C07980=1025.986,-15.091,405.957,167.347,46.507,158.566
C07981=1025.980,-15.341,405.971,167.344,46.510,158.567
C07982=1025.974,-15.590,405.984,167.342,46.512,158.567
C07983=1025.968,-15.840,405.998,167.339,46.515,158.567
C07984=1025.962,-16.089,406.012,167.336,46.517,158.567
C07985=1025.955,-16.339,406.025,167.333,46.521,158.567
C07986=1025.950,-16.590,406.038,167.331,46.523,158.568
C07987=1025.943,-16.839,406.052,167.328,46.526,158.568
C07988=1025.937,-17.088,406.065,167.325,46.529,158.568
C07989=1025.931,-17.337,406.078,167.322,46.532,158.568
C07990=1025.925,-17.588,406.092,167.320,46.535,158.568
C07991=1025.919,-17.837,406.106,167.318,46.538,158.569
C07992=1025.912,-18.086,406.119,167.314,46.540,158.569
C07993=1025.906,-18.335,406.132,167.312,46.543,158.569
C07994=1025.900,-18.586,406.146,167.309,46.546,158.569
C07995=1025.894,-18.835,406.160,167.306,46.549,158.569
C07996=1025.888,-19.084,406.173,167.303,46.552,158.569
C07997=1025.882,-19.334,406.186,167.301,46.555,158.570
C07998=1025.876,-19.584,406.199,167.298,46.557,158.570
C07999=1025.870,-19.834,406.213,167.295,46.560,158.570
C08000=1025.863,-20.083,406.226,167.293,46.562,158.570
C08001=1025.856,-20.363,406.241,167.289,46.565,158.570
C08002=1025.849,-20.644,406.257,167.286,46.569,158.570
C08003=1025.843,-20.925,406.271,167.283,46.572,158.571
C08004=1025.836,-21.205,406.286,167.280,46.575,158.571
C08005=1025.829,-21.455,406.300,167.278,46.578,158.571
C08006=1025.823,-21.705,406.313,167.274,46.580,158.571
C08007=1025.818,-21.955,406.326,167.272,46.583,158.571
C08008=1025.812,-22.204,406.340,167.269,46.586,158.572
C08009=1025.806,-22.453,406.353,167.266,46.589,158.572
C08010=1025.799,-22.702,406.366,167.264,46.592,158.572
C08011=1025.794,-22.953,406.379,167.261,46.594,158.572
C08012=1025.787,-23.203,406.393,167.258,46.597,158.572
C08013=1025.781,-23.452,406.406,167.255,46.600,158.572
C08014=1025.775,-23.701,406.419,167.253,46.603,158.573
C08015=1025.769,-23.951,406.432,167.250,46.606,158.573
C08016=1025.764,-24.201,406.446,167.247,46.608,158.573
C08017=1025.757,-24.450,406.459,167.245,46.611,158.573
C08018=1025.751,-24.699,406.472,167.242,46.614,158.573
C08019=1025.745,-24.949,406.485,167.239,46.617,158.574
C08020=1025.739,-25.198,406.498,167.236,46.619,158.574
C08021=1025.734,-25.448,406.512,167.234,46.622,158.574
C08022=1025.728,-25.698,406.525,167.230,46.625,158.574
C08023=1025.721,-25.948,406.538,167.228,46.628,158.574
C08024=1025.715,-26.197,406.552,167.226,46.630,158.574
C08025=1025.710,-26.447,406.565,167.222,46.633,158.574
C08026=1025.703,-26.696,406.578,167.220,46.636,158.575
C08027=1025.697,-26.946,406.591,167.217,46.639,158.575
C08028=1025.691,-27.196,406.604,167.214,46.641,158.575
C08029=1025.685,-27.445,406.617,167.211,46.644,158.575
C08030=1025.679,-27.695,406.630,167.209,46.647,158.575
C08031=1025.673,-27.944,406.643,167.206,46.650,158.576
C08032=1025.667,-28.194,406.655,167.203,46.652,158.576
C08033=1025.661,-28.443,406.669,167.200,46.655,158.576
C08034=1025.655,-28.693,406.681,167.198,46.658,158.576
C08035=1025.649,-28.942,406.695,167.195,46.661,158.576
C08036=1025.643,-29.192,406.707,167.192,46.663,158.576
C08037=1025.636,-29.441,406.720,167.189,46.666,158.577
C08038=1025.631,-29.691,406.733,167.187,46.669,158.577
C08039=1025.624,-29.941,406.746,167.183,46.672,158.577
C08040=1025.618,-30.190,406.759,167.181,46.675,158.577
C08041=1025.612,-30.440,406.772,167.178,46.678,158.577
C08042=1025.606,-30.689,406.784,167.176,46.681,158.578
C08043=1025.599,-30.939,406.797,167.172,46.684,158.578
C08044=1025.593,-31.188,406.810,167.170,46.686,158.578
C08045=1025.588,-31.438,406.822,167.167,46.689,158.578
C08046=1025.581,-31.688,406.836,167.164,46.692,158.578
C08047=1025.575,-31.937,406.848,167.161,46.695,158.578
C08048=1025.569,-32.187,406.861,167.159,46.698,158.579
C08049=1025.563,-32.437,406.874,167.156,46.701,158.579
C08050=1025.557,-32.687,406.887,167.153,46.704,158.579
C08051=1025.551,-32.936,406.900,167.150,46.706,158.579
C08052=1025.545,-33.186,406.912,167.148,46.709,158.579
C08053=1025.539,-33.436,406.925,167.144,46.712,158.579
C08054=1025.533,-33.685,406.938,167.142,46.715,158.580
C08055=1025.527,-33.935,406.951,167.139,46.718,158.580
C08056=1025.521,-34.184,406.963,167.137,46.721,158.580
C08057=1025.514,-34.434,406.976,167.133,46.723,158.580
C08058=1025.508,-34.683,406.989,167.131,46.726,158.580
C08059=1025.503,-34.933,407.001,167.128,46.729,158.580
C08060=1025.496,-35.183,407.014,167.125,46.732,158.581
C08061=1025.491,-35.432,407.027,167.122,46.735,158.581
C08062=1025.485,-35.682,407.039,167.120,46.737,158.581
C08063=1025.479,-35.932,407.052,167.116,46.740,158.581
C08064=1025.473,-36.181,407.065,167.114,46.743,158.581
C08065=1025.466,-36.460,407.078,167.111,46.746,158.581
C08066=1025.459,-36.741,407.093,167.108,46.749,158.582
C08067=1025.453,-37.020,407.107,167.104,46.752,158.582
C08068=1025.446,-37.300,407.121,167.101,46.756,158.582
C08069=1025.441,-37.550,407.133,167.098,46.758,158.582
C08070=1025.434,-37.799,407.147,167.096,46.761,158.582
C08071=1025.428,-38.049,407.159,167.092,46.764,158.582
C08072=1025.422,-38.299,407.171,167.090,46.767,158.583
C08073=1025.416,-38.548,407.184,167.086,46.769,158.583
C08074=1025.410,-38.798,407.196,167.084,46.772,158.583
C08075=1025.404,-39.047,407.209,167.081,46.775,158.583
C08076=1025.398,-39.297,407.222,167.079,46.778,158.583
C08077=1025.392,-39.547,407.234,167.076,46.781,158.583
C08078=1025.386,-39.796,407.246,167.073,46.783,158.584
C08079=1025.380,-40.046,407.259,167.070,46.787,158.584
C08080=1025.373,-40.296,407.271,167.067,46.790,158.584
C08081=1025.367,-40.546,407.283,167.064,46.792,158.584
C08082=1025.362,-40.795,407.296,167.061,46.795,158.584
C08083=1025.355,-41.044,407.308,167.059,46.798,158.584
C08084=1025.350,-41.294,407.320,167.056,46.801,158.585
C08085=1025.344,-41.544,407.333,167.053,46.803,158.585
C08086=1025.337,-41.794,407.345,167.050,46.807,158.585
C08087=1025.332,-42.043,407.357,167.047,46.810,158.585
C08088=1025.326,-42.293,407.369,167.045,46.812,158.585
C08089=1025.319,-42.542,407.381,167.041,46.815,158.585
C08090=1025.313,-42.792,407.394,167.039,46.818,158.586
C08091=1025.307,-43.041,407.405,167.036,46.821,158.586
C08092=1025.301,-43.291,407.418,167.033,46.823,158.586
C08093=1025.295,-43.541,407.431,167.030,46.827,158.586
C08094=1025.289,-43.790,407.443,167.027,46.830,158.586
C08095=1025.283,-44.040,407.455,167.025,46.832,158.586
C08096=1025.277,-44.289,407.467,167.021,46.836,158.587
C08097=1025.271,-44.539,407.479,167.019,46.838,158.587
C08098=1025.265,-44.789,407.491,167.016,46.841,158.587
C08099=1025.259,-45.038,407.503,167.013,46.844,158.587
C08100=1025.253,-45.288,407.515,167.010,46.847,158.587
C08101=1025.247,-45.538,407.528,167.007,46.850,158.587
C08102=1025.241,-45.788,407.540,167.005,46.852,158.588
C08103=1025.235,-46.037,407.552,167.001,46.856,158.588
C08104=1025.229,-46.286,407.564,166.999,46.858,158.588
C08105=1025.223,-46.536,407.576,166.996,46.861,158.588
C08106=1025.218,-46.786,407.588,166.993,46.864,158.588
C08107=1025.211,-47.036,407.600,166.990,46.867,158.588
C08108=1025.205,-47.286,407.612,166.987,46.870,158.588
C08109=1025.199,-47.534,407.624,166.985,46.873,158.589
C08110=1025.193,-47.784,407.637,166.981,46.876,158.589
C08111=1025.187,-48.034,407.649,166.979,46.878,158.589
C08112=1025.182,-48.284,407.660,166.976,46.881,158.589
C08113=1025.176,-48.534,407.673,166.972,46.884,158.589
C08114=1025.169,-48.783,407.684,166.970,46.887,158.589
C08115=1025.164,-49.032,407.697,166.967,46.890,158.590
C08116=1025.158,-49.283,407.709,166.965,46.893,158.590
C08117=1025.152,-49.532,407.720,166.961,46.896,158.590
C08118=1025.146,-49.782,407.733,166.959,46.898,158.590
C08119=1025.140,-50.031,407.745,166.956,46.901,158.590
C08120=1025.135,-50.281,407.756,166.952,46.904,158.590
C08121=1025.129,-50.531,407.769,166.950,46.907,158.591
C08122=1025.122,-50.780,407.781,166.947,46.910,158.591
C08123=1025.117,-51.030,407.792,166.945,46.913,158.591
C08124=1025.110,-51.280,407.804,166.941,46.916,158.591
C08125=1025.104,-51.529,407.816,166.938,46.919,158.591
C08126=1025.098,-51.779,407.827,166.935,46.922,158.591
C08127=1025.091,-52.028,407.839,166.933,46.925,158.592
C08128=1025.086,-52.278,407.850,166.929,46.928,158.592
C08129=1025.078,-52.582,407.864,166.926,46.932,158.592
C08130=1025.071,-52.886,407.879,166.922,46.936,158.592
C08131=1025.064,-53.190,407.892,166.919,46.939,158.592
C08132=1025.056,-53.494,407.907,166.915,46.943,158.593
C08133=1025.050,-53.744,407.918,166.912,46.946,158.593
C08134=1025.044,-53.993,407.930,166.910,46.949,158.593
C08135=1025.038,-54.243,407.941,166.906,46.952,158.593
C08136=1025.032,-54.492,407.953,166.903,46.955,158.593
C08137=1025.026,-54.742,407.964,166.901,46.958,158.594
C08138=1025.019,-54.992,407.976,166.898,46.961,158.594
C08139=1025.013,-55.241,407.987,166.894,46.964,158.594
C08140=1025.007,-55.491,408.000,166.892,46.967,158.594
C08141=1025.002,-55.741,408.011,166.889,46.970,158.594
C08142=1024.995,-55.991,408.022,166.886,46.973,158.594
C08143=1024.989,-56.240,408.033,166.883,46.976,158.595
C08144=1024.983,-56.490,408.045,166.880,46.979,158.595
C08145=1024.978,-56.739,408.057,166.877,46.982,158.595
C08146=1024.971,-56.989,408.068,166.874,46.985,158.595
C08147=1024.966,-57.239,408.079,166.872,46.988,158.595
C08148=1024.959,-57.489,408.091,166.868,46.991,158.595
C08149=1024.953,-57.738,408.102,166.865,46.994,158.596
C08150=1024.947,-57.988,408.114,166.863,46.997,158.596
C08151=1024.942,-58.237,408.125,166.860,47.000,158.596
C08152=1024.935,-58.488,408.136,166.856,47.003,158.596
C08153=1024.929,-58.736,408.148,166.854,47.006,158.596
C08154=1024.923,-58.987,408.159,166.851,47.009,158.596
C08155=1024.917,-59.236,408.170,166.848,47.012,158.597
C08156=1024.911,-59.487,408.182,166.845,47.015,158.597
C08157=1024.905,-59.736,408.194,166.842,47.018,158.597
C08158=1024.900,-59.985,408.204,166.839,47.021,158.597
C08159=1024.893,-60.235,408.216,166.837,47.024,158.597
C08160=1024.887,-60.484,408.227,166.833,47.027,158.597
C08161=1024.881,-60.734,408.239,166.830,47.030,158.598
C08162=1024.876,-60.984,408.250,166.828,47.033,158.598
C08163=1024.870,-61.234,408.261,166.825,47.036,158.598
C08164=1024.864,-61.483,408.273,166.821,47.039,158.598
C08165=1024.858,-61.733,408.284,166.818,47.042,158.598
C08166=1024.852,-61.983,408.295,166.816,47.045,158.598
C08167=1024.846,-62.232,408.306,166.813,47.048,158.599
C08168=1024.840,-62.481,408.318,166.809,47.051,158.599
C08169=1024.834,-62.720,408.329,166.807,47.054,158.599
C08170=1024.828,-62.958,408.339,166.804,47.056,158.599
C08171=1024.823,-63.195,408.349,166.801,47.059,158.599
C08172=1024.818,-63.434,408.361,166.798,47.062,158.599
C08173=1024.812,-63.671,408.371,166.796,47.065,158.600
C08174=1024.806,-63.909,408.382,166.793,47.068,158.600
C08175=1024.801,-64.146,408.393,166.790,47.070,158.600
C08176=1024.795,-64.384,408.403,166.787,47.073,158.600
C08177=1024.789,-64.634,408.414,166.785,47.076,158.600
C08178=1024.784,-64.883,408.425,166.782,47.079,158.600
C08179=1024.777,-65.134,408.436,166.778,47.082,158.600
C08180=1024.772,-65.383,408.448,166.776,47.085,158.601
C08181=1024.766,-65.633,408.459,166.773,47.088,158.601
C08182=1024.760,-65.882,408.471,166.770,47.091,158.601
C08183=1024.754,-66.132,408.482,166.767,47.093,158.601
C08184=1024.748,-66.381,408.492,166.764,47.097,158.601
C08185=1024.742,-66.632,408.504,166.761,47.100,158.601
C08186=1024.736,-66.881,408.515,166.758,47.103,158.601
C08187=1024.730,-67.131,408.525,166.755,47.106,158.602
C08188=1024.725,-67.380,408.537,166.752,47.109,158.602
C08189=1024.719,-67.631,408.548,166.750,47.112,158.602
C08190=1024.713,-67.880,408.559,166.746,47.115,158.602
C08191=1024.708,-68.130,408.570,166.743,47.118,158.602
C08192=1024.702,-68.379,408.581,166.741,47.120,158.602
C08193=1024.696,-68.661,408.593,166.737,47.124,158.602
C08194=1024.689,-68.942,408.606,166.733,47.127,158.603
C08195=1024.682,-69.223,408.618,166.730,47.130,158.603
C08196=1024.676,-69.505,408.631,166.727,47.133,158.603
C08197=1024.670,-69.754,408.641,166.724,47.136,158.603
C08198=1024.664,-70.005,408.653,166.721,47.139,158.603
C08199=1024.658,-70.254,408.664,166.718,47.142,158.603
C08200=1024.653,-70.504,408.674,166.715,47.145,158.604
C08201=1024.647,-70.753,408.685,166.713,47.148,158.604
C08202=1024.641,-71.003,408.696,166.709,47.151,158.604
C08203=1024.636,-71.253,408.708,166.706,47.154,158.604
C08204=1024.630,-71.503,408.719,166.704,47.157,158.604
C08205=1024.624,-71.752,408.730,166.700,47.160,158.604
C08206=1024.618,-72.002,408.741,166.697,47.163,158.604
C08207=1024.613,-72.251,408.752,166.695,47.166,158.605
C08208=1024.607,-72.501,408.762,166.692,47.169,158.605
C08209=1024.601,-72.750,408.773,166.688,47.171,158.605
C08210=1024.595,-73.001,408.784,166.686,47.174,158.605
C08211=1024.589,-73.250,408.795,166.683,47.177,158.605
C08212=1024.584,-73.500,408.806,166.680,47.180,158.605
C08213=1024.579,-73.750,408.817,166.677,47.183,158.605
C08214=1024.573,-73.999,408.828,166.674,47.186,158.606
C08215=1024.567,-74.249,408.839,166.671,47.189,158.605
C08216=1024.562,-74.499,408.849,166.668,47.191,158.606
C08217=1024.555,-74.749,408.860,166.665,47.195,158.606
C08218=1024.549,-74.998,408.870,166.662,47.198,158.606
C08219=1024.543,-75.248,408.881,166.659,47.201,158.606
C08220=1024.538,-75.498,408.891,166.655,47.204,158.606
C08221=1024.532,-75.747,408.902,166.653,47.207,158.606
C08222=1024.526,-75.997,408.913,166.650,47.210,158.607
C08223=1024.520,-76.246,408.923,166.647,47.213,158.607
C08224=1024.514,-76.496,408.934,166.643,47.216,158.607
C08225=1024.509,-76.746,408.944,166.641,47.219,158.607
C08226=1024.503,-76.996,408.955,166.638,47.222,158.607
C08227=1024.497,-77.246,408.966,166.635,47.225,158.607
C08228=1024.491,-77.496,408.976,166.631,47.228,158.607
C08229=1024.485,-77.745,408.986,166.629,47.231,158.608
C08230=1024.479,-77.995,408.997,166.626,47.234,158.608
C08231=1024.474,-78.245,409.007,166.623,47.237,158.608
C08232=1024.468,-78.494,409.018,166.619,47.240,158.608
C08233=1024.462,-78.744,409.028,166.617,47.243,158.608
C08234=1024.456,-78.993,409.039,166.614,47.246,158.608
C08235=1024.451,-79.244,409.049,166.611,47.249,158.609
C08236=1024.445,-79.493,409.060,166.608,47.253,158.609
C08237=1024.439,-79.743,409.070,166.605,47.255,158.609
C08238=1024.433,-79.992,409.080,166.602,47.259,158.609
C08239=1024.428,-80.242,409.090,166.599,47.262,158.609
C08240=1024.422,-80.492,409.101,166.596,47.266,158.609
C08241=1024.416,-80.742,409.111,166.594,47.268,158.610
C08242=1024.410,-80.991,409.122,166.590,47.271,158.610
C08243=1024.404,-81.241,409.131,166.587,47.275,158.610
C08244=1024.398,-81.490,409.142,166.584,47.278,158.610
C08245=1024.392,-81.740,409.152,166.581,47.281,158.610
C08246=1024.386,-81.990,409.162,166.577,47.284,158.610
C08247=1024.380,-82.240,409.172,166.576,47.288,158.611
C08248=1024.374,-82.490,409.182,166.572,47.291,158.611
C08249=1024.368,-82.739,409.192,166.569,47.294,158.611
C08250=1024.363,-82.989,409.203,166.566,47.297,158.611
C08251=1024.356,-83.239,409.212,166.563,47.300,158.611
C08252=1024.351,-83.489,409.223,166.559,47.303,158.611
C08253=1024.344,-83.738,409.233,166.557,47.306,158.612
C08254=1024.339,-83.988,409.243,166.554,47.310,158.612
C08255=1024.333,-84.238,409.253,166.551,47.313,158.612
C08256=1024.327,-84.487,409.263,166.548,47.316,158.612
C08257=1024.320,-84.771,409.274,166.544,47.319,158.612
C08258=1024.314,-85.055,409.286,166.540,47.323,158.612
C08259=1024.308,-85.337,409.297,166.537,47.326,158.613
C08260=1024.301,-85.621,409.309,166.534,47.330,158.613
C08261=1024.295,-85.871,409.318,166.531,47.333,158.613
C08262=1024.290,-86.121,409.329,166.528,47.336,158.613
C08263=1024.283,-86.370,409.339,166.525,47.340,158.613
C08264=1024.278,-86.620,409.349,166.522,47.342,158.613
C08265=1024.272,-86.870,409.359,166.519,47.346,158.614
C08266=1024.266,-87.120,409.369,166.516,47.349,158.614
C08267=1024.260,-87.370,409.378,166.513,47.352,158.614
C08268=1024.255,-87.619,409.389,166.510,47.356,158.614
C08269=1024.249,-87.869,409.398,166.506,47.359,158.614
C08270=1024.243,-88.119,409.409,166.504,47.362,158.614
C08271=1024.237,-88.369,409.418,166.501,47.365,158.615
C08272=1024.232,-88.619,409.428,166.498,47.368,158.615
C08273=1024.225,-88.868,409.439,166.495,47.371,158.615
C08274=1024.220,-89.117,409.448,166.491,47.374,158.615
C08275=1024.214,-89.367,409.458,166.489,47.377,158.615
C08276=1024.209,-89.617,409.468,166.486,47.380,158.615
C08277=1024.203,-89.867,409.478,166.483,47.384,158.616
C08278=1024.197,-90.117,409.488,166.480,47.387,158.616
C08279=1024.192,-90.366,409.497,166.476,47.390,158.616
C08280=1024.185,-90.616,409.507,166.474,47.393,158.616
C08281=1024.180,-90.866,409.517,166.471,47.396,158.616
C08282=1024.174,-91.115,409.527,166.468,47.399,158.616
C08283=1024.169,-91.365,409.537,166.464,47.402,158.616
C08284=1024.163,-91.614,409.546,166.461,47.406,158.616
C08285=1024.157,-91.865,409.557,166.459,47.408,158.617
C08286=1024.151,-92.114,409.566,166.456,47.412,158.617
C08287=1024.146,-92.364,409.576,166.453,47.415,158.617
C08288=1024.140,-92.614,409.585,166.449,47.418,158.617
C08289=1024.135,-92.864,409.596,166.446,47.421,158.617
C08290=1024.128,-93.113,409.605,166.444,47.424,158.617
C08291=1024.124,-93.363,409.615,166.441,47.427,158.618
C08292=1024.117,-93.613,409.625,166.437,47.430,158.618
C08293=1024.112,-93.863,409.635,166.434,47.433,158.618
C08294=1024.106,-94.113,409.644,166.431,47.436,158.618
C08295=1024.101,-94.362,409.654,166.429,47.439,158.618
C08296=1024.095,-94.612,409.664,166.426,47.443,158.618
C08297=1024.089,-94.862,409.673,166.423,47.446,158.619
C08298=1024.084,-95.111,409.683,166.419,47.449,158.619
C08299=1024.078,-95.361,409.693,166.416,47.452,158.619
C08300=1024.072,-95.611,409.703,166.414,47.455,158.619
C08301=1024.067,-95.860,409.712,166.411,47.458,158.619
C08302=1024.061,-96.111,409.721,166.407,47.462,158.619
C08303=1024.055,-96.361,409.731,166.404,47.465,158.619
C08304=1024.050,-96.610,409.741,166.401,47.468,158.619
C08305=1024.044,-96.860,409.750,166.399,47.471,158.620
C08306=1024.039,-97.109,409.760,166.395,47.474,158.620
C08307=1024.033,-97.359,409.770,166.392,47.477,158.620
C08308=1024.027,-97.609,409.779,166.389,47.480,158.620
C08309=1024.022,-97.858,409.789,166.386,47.483,158.620
C08310=1024.016,-98.109,409.798,166.384,47.486,158.620
C08311=1024.010,-98.358,409.807,166.380,47.489,158.620
C08312=1024.005,-98.607,409.817,166.377,47.492,158.621
C08313=1023.998,-98.857,409.826,166.374,47.496,158.621
C08314=1023.994,-99.107,409.835,166.371,47.499,158.621
C08315=1023.988,-99.357,409.845,166.368,47.503,158.621
C08316=1023.982,-99.607,409.854,166.364,47.506,158.621
C08317=1023.976,-99.857,409.863,166.361,47.509,158.621
C08318=1023.970,-100.106,409.873,166.359,47.512,158.622
C08319=1023.965,-100.355,409.882,166.356,47.516,158.622
C08320=1023.959,-100.606,409.891,166.353,47.519,158.622
C08321=1023.952,-100.891,409.902,166.349,47.523,158.622
C08322=1023.946,-101.177,409.912,166.346,47.526,158.622
C08323=1023.940,-101.462,409.924,166.343,47.530,158.623
C08324=1023.933,-101.748,409.933,166.338,47.533,158.623
C08325=1023.928,-101.999,409.943,166.335,47.537,158.623
C08326=1023.922,-102.248,409.952,166.332,47.540,158.623
C08327=1023.916,-102.498,409.962,166.330,47.543,158.623
C08328=1023.911,-102.747,409.970,166.327,47.546,158.623
C08329=1023.905,-102.997,409.980,166.324,47.549,158.623
C08330=1023.899,-103.247,409.988,166.320,47.553,158.623
C08331=1023.893,-103.497,409.998,166.317,47.556,158.624
C08332=1023.888,-103.746,410.008,166.314,47.560,158.624
C08333=1023.883,-103.996,410.016,166.311,47.563,158.624
C08334=1023.877,-104.246,410.026,166.309,47.566,158.624
C08335=1023.871,-104.496,410.034,166.306,47.569,158.624
C08336=1023.866,-104.745,410.044,166.302,47.572,158.624
C08337=1023.860,-104.995,410.052,166.299,47.576,158.625
C08338=1023.854,-105.245,410.062,166.296,47.579,158.625
C08339=1023.849,-105.495,410.071,166.293,47.582,158.625
C08340=1023.843,-105.744,410.080,166.290,47.585,158.625
C08341=1023.838,-105.995,410.089,166.287,47.588,158.625
C08342=1023.832,-106.244,410.098,166.284,47.591,158.625
C08343=1023.826,-106.494,410.107,166.281,47.595,158.626
C08344=1023.820,-106.743,410.116,166.278,47.598,158.626
C08345=1023.815,-106.993,410.125,166.275,47.601,158.626
C08346=1023.809,-107.244,410.134,166.272,47.605,158.626
C08347=1023.804,-107.493,410.143,166.268,47.608,158.626
C08348=1023.798,-107.743,410.152,166.265,47.611,158.626
C08349=1023.792,-107.992,410.161,166.263,47.614,158.627
C08350=1023.786,-108.243,410.170,166.260,47.618,158.627
C08351=1023.781,-108.492,410.178,166.257,47.621,158.627
C08352=1023.776,-108.741,410.188,166.254,47.624,158.627
C08353=1023.770,-108.992,410.196,166.251,47.628,158.627
C08354=1023.765,-109.242,410.205,166.247,47.631,158.627
C08355=1023.758,-109.491,410.214,166.244,47.634,158.627
C08356=1023.753,-109.741,410.223,166.241,47.637,158.628
C08357=1023.748,-109.991,410.231,166.238,47.641,158.628
C08358=1023.742,-110.241,410.241,166.236,47.644,158.628
C08359=1023.736,-110.490,410.249,166.233,47.647,158.628
C08360=1023.731,-110.740,410.258,166.229,47.650,158.628
C08361=1023.725,-110.990,410.267,166.226,47.654,158.629
C08362=1023.720,-111.239,410.276,166.223,47.657,158.629
C08363=1023.714,-111.489,410.284,166.220,47.661,158.629
C08364=1023.708,-111.739,410.293,166.217,47.664,158.629
C08365=1023.703,-111.989,410.301,166.214,47.668,158.629
C08366=1023.697,-112.238,410.310,166.211,47.671,158.629
C08367=1023.691,-112.489,410.319,166.208,47.674,158.629
C08368=1023.686,-112.738,410.328,166.205,47.677,158.630
C08369=1023.681,-112.988,410.336,166.202,47.680,158.630
C08370=1023.675,-113.238,410.345,166.199,47.684,158.630
C08371=1023.669,-113.487,410.354,166.196,47.687,158.630
C08372=1023.664,-113.737,410.363,166.192,47.690,158.630
C08373=1023.658,-113.988,410.372,166.189,47.693,158.630
C08374=1023.653,-114.237,410.380,166.186,47.697,158.631
C08375=1023.647,-114.487,410.389,166.183,47.700,158.631
C08376=1023.641,-114.736,410.397,166.181,47.703,158.631
C08377=1023.636,-114.987,410.405,166.178,47.706,158.631
C08378=1023.630,-115.237,410.414,166.175,47.710,158.631
C08379=1023.625,-115.486,410.422,166.171,47.713,158.631
C08380=1023.620,-115.735,410.432,166.168,47.717,158.631
C08381=1023.613,-115.985,410.440,166.165,47.720,158.632
C08382=1023.608,-116.235,410.448,166.162,47.724,158.632
C08383=1023.602,-116.485,410.457,166.159,47.727,158.632
C08384=1023.597,-116.735,410.465,166.156,47.730,158.632
C08385=1023.590,-117.020,410.475,166.153,47.734,158.632
C08386=1023.584,-117.306,410.484,166.149,47.738,158.632
C08387=1023.577,-117.591,410.494,166.146,47.742,158.633
C08388=1023.571,-117.876,410.503,166.142,47.745,158.633
C08389=1023.566,-118.126,410.512,166.140,47.749,158.633
C08390=1023.561,-118.376,410.520,166.136,47.752,158.633
C08391=1023.555,-118.625,410.529,166.133,47.755,158.633
C08392=1023.549,-118.875,410.537,166.130,47.759,158.634
C08393=1023.544,-119.125,410.546,166.127,47.762,158.634
C08394=1023.538,-119.375,410.554,166.124,47.765,158.634
C08395=1023.533,-119.625,410.563,166.121,47.769,158.634
C08396=1023.527,-119.874,410.571,166.118,47.772,158.634
C08397=1023.522,-120.124,410.578,166.114,47.776,158.634
C08398=1023.516,-120.375,410.587,166.111,47.779,158.634
C08399=1023.510,-120.624,410.595,166.108,47.783,158.635
C08400=1023.505,-120.874,410.604,166.106,47.786,158.635
C08401=1023.500,-121.124,410.612,166.103,47.789,158.635
C08402=1023.494,-121.373,410.620,166.100,47.792,158.635
C08403=1023.488,-121.623,410.628,166.097,47.796,158.635
C08404=1023.483,-121.873,410.636,166.094,47.799,158.635
C08405=1023.478,-122.123,410.645,166.090,47.802,158.636
C08406=1023.472,-122.373,410.653,166.087,47.806,158.636
C08407=1023.466,-122.623,410.661,166.084,47.809,158.636
C08408=1023.461,-122.872,410.670,166.081,47.812,158.636
C08409=1023.455,-123.122,410.678,166.078,47.816,158.636
C08410=1023.450,-123.372,410.686,166.076,47.819,158.636
C08411=1023.445,-123.622,410.694,166.073,47.822,158.637
C08412=1023.439,-123.871,410.702,166.069,47.826,158.637
C08413=1023.434,-124.121,410.710,166.066,47.829,158.637
C08414=1023.429,-124.371,410.718,166.063,47.833,158.637
C08415=1023.423,-124.621,410.726,166.060,47.836,158.637
C08416=1023.417,-124.870,410.735,166.057,47.840,158.637
C08417=1023.412,-125.121,410.742,166.054,47.843,158.637
C08418=1023.406,-125.370,410.750,166.051,47.846,158.638
C08419=1023.401,-125.620,410.759,166.048,47.850,158.638
C08420=1023.395,-125.870,410.766,166.044,47.853,158.638
C08421=1023.390,-126.119,410.774,166.042,47.857,158.638
C08422=1023.384,-126.369,410.782,166.038,47.860,158.638
C08423=1023.379,-126.619,410.790,166.036,47.863,158.639
C08424=1023.373,-126.869,410.798,166.033,47.867,158.639
C08425=1023.368,-127.118,410.806,166.030,47.870,158.639
C08426=1023.362,-127.368,410.814,166.027,47.873,158.639
C08427=1023.357,-127.618,410.822,166.024,47.877,158.639
C08428=1023.351,-127.868,410.829,166.021,47.880,158.639
C08429=1023.346,-128.118,410.838,166.017,47.884,158.639
C08430=1023.341,-128.368,410.847,166.015,47.886,158.640
C08431=1023.337,-128.617,410.856,166.012,47.889,158.640
C08432=1023.333,-128.867,410.866,166.009,47.890,158.639
C08433=1023.331,-129.116,410.876,166.006,47.892,158.639
C08434=1023.327,-129.366,410.887,166.004,47.892,158.639
C08435=1023.325,-129.616,410.899,166.002,47.892,158.639
C08436=1023.324,-129.865,410.911,165.999,47.892,158.638
C08437=1023.323,-130.115,410.924,165.997,47.891,158.638
C08438=1023.321,-130.365,410.938,165.994,47.890,158.637
C08439=1023.321,-130.615,410.952,165.992,47.888,158.637
C08440=1023.322,-130.864,410.966,165.990,47.886,158.636
C08441=1023.323,-131.114,410.980,165.987,47.883,158.635
C08442=1023.324,-131.364,410.996,165.986,47.880,158.635
C08443=1023.325,-131.614,411.013,165.984,47.876,158.634
C08444=1023.329,-131.864,411.029,165.983,47.872,158.633
C08445=1023.332,-132.114,411.048,165.981,47.867,158.632
C08446=1023.335,-132.364,411.065,165.980,47.862,158.631
C08447=1023.339,-132.613,411.084,165.978,47.856,158.630
C08448=1023.343,-132.863,411.103,165.977,47.850,158.628
C08449=1023.051,-132.889,410.762,165.929,48.138,158.670
C08450=1023.046,-132.639,410.742,165.930,48.144,158.671
C08451=1023.042,-132.390,410.725,165.931,48.150,158.673
C08452=1023.039,-132.139,410.706,165.934,48.155,158.674
C08453=1023.036,-131.890,410.689,165.934,48.160,158.675
C08454=1023.034,-131.640,410.671,165.936,48.164,158.676
C08455=1023.031,-131.390,410.655,165.938,48.168,158.676
C08456=1023.030,-131.140,410.640,165.940,48.171,158.677
C08457=1023.030,-130.891,410.625,165.943,48.174,158.678
C08458=1023.029,-130.640,410.610,165.945,48.176,158.679
C08459=1023.030,-130.391,410.596,165.947,48.178,158.680
C08460=1023.030,-130.141,410.582,165.949,48.179,158.680
C08461=1023.031,-129.891,410.570,165.951,48.180,158.680
C08462=1023.032,-129.642,410.558,165.954,48.180,158.681
C08463=1023.035,-129.392,410.546,165.956,48.180,158.681
C08464=1023.037,-129.142,410.535,165.959,48.179,158.681
C08465=1023.041,-128.893,410.525,165.962,48.178,158.681
C08466=1023.044,-128.643,410.514,165.965,48.176,158.682
C08467=1023.048,-128.393,410.505,165.967,48.174,158.682
C08468=1023.053,-128.144,410.497,165.971,48.171,158.682
C08469=1023.058,-127.894,410.488,165.973,48.168,158.681
C08470=1023.064,-127.644,410.480,165.976,48.164,158.681
C08471=1023.069,-127.394,410.473,165.979,48.161,158.681
C08472=1023.075,-127.145,410.464,165.982,48.157,158.681
C08473=1023.080,-126.895,410.457,165.985,48.154,158.681
C08474=1023.086,-126.645,410.449,165.988,48.150,158.680
C08475=1023.092,-126.396,410.441,165.991,48.147,158.680
C08476=1023.097,-126.145,410.433,165.994,48.144,158.680
C08477=1023.103,-125.896,410.425,165.997,48.140,158.680
C08478=1023.108,-125.646,410.417,166.000,48.137,158.680
C08479=1023.114,-125.396,410.409,166.003,48.133,158.680
C08480=1023.119,-125.146,410.401,166.006,48.130,158.680
C08481=1023.124,-124.896,410.393,166.010,48.126,158.679
C08482=1023.130,-124.647,410.385,166.013,48.122,158.679
C08483=1023.135,-124.397,410.377,166.016,48.119,158.679
C08484=1023.141,-124.147,410.370,166.019,48.115,158.679
C08485=1023.146,-123.897,410.361,166.022,48.112,158.679
C08486=1023.151,-123.647,410.353,166.025,48.109,158.679
C08487=1023.157,-123.398,410.345,166.028,48.105,158.678
C08488=1023.162,-123.148,410.337,166.031,48.102,158.678
C08489=1023.167,-122.898,410.328,166.034,48.099,158.678
C08490=1023.173,-122.649,410.321,166.036,48.095,158.678
C08491=1023.179,-122.399,410.312,166.039,48.092,158.678
C08492=1023.184,-122.149,410.304,166.043,48.089,158.678
C08493=1023.189,-121.899,410.296,166.046,48.085,158.677
C08494=1023.196,-121.649,410.288,166.049,48.081,158.677
C08495=1023.201,-121.399,410.279,166.052,48.078,158.677
C08496=1023.206,-121.149,410.271,166.055,48.074,158.677
C08497=1023.212,-120.900,410.263,166.058,48.071,158.677
C08498=1023.217,-120.650,410.255,166.061,48.067,158.677
C08499=1023.222,-120.400,410.246,166.064,48.064,158.676
C08500=1023.228,-120.150,410.238,166.067,48.061,158.676
C08501=1023.234,-119.901,410.230,166.070,48.057,158.676
C08502=1023.239,-119.651,410.222,166.074,48.054,158.676
C08503=1023.245,-119.401,410.213,166.077,48.051,158.676
C08504=1023.251,-119.151,410.205,166.080,48.047,158.676
C08505=1023.256,-118.901,410.196,166.083,48.043,158.676
C08506=1023.261,-118.652,410.188,166.086,48.040,158.675
C08507=1023.267,-118.402,410.179,166.089,48.036,158.675
C08508=1023.272,-118.152,410.172,166.092,48.033,158.675
C08509=1023.278,-117.902,410.163,166.094,48.030,158.675
C08510=1023.284,-117.617,410.154,166.098,48.026,158.675
C08511=1023.291,-117.332,410.144,166.101,48.022,158.674
C08512=1023.297,-117.047,410.135,166.105,48.018,158.674
C08513=1023.303,-116.761,410.124,166.108,48.014,158.674
C08514=1023.309,-116.512,410.116,166.111,48.011,158.674
C08515=1023.314,-116.262,410.108,166.114,48.008,158.674
C08516=1023.319,-116.012,410.099,166.117,48.004,158.673
C08517=1023.325,-115.762,410.091,166.121,48.001,158.673
C08518=1023.331,-115.512,410.082,166.124,47.997,158.673
C08519=1023.337,-115.263,410.074,166.127,47.994,158.673
C08520=1023.342,-115.013,410.066,166.130,47.990,158.673
C08521=1023.348,-114.763,410.057,166.133,47.986,158.673
C08522=1023.353,-114.513,410.048,166.136,47.983,158.673
C08523=1023.358,-114.263,410.040,166.139,47.980,158.672
C08524=1023.364,-114.013,410.031,166.142,47.977,158.672
C08525=1023.370,-113.763,410.023,166.145,47.973,158.672
C08526=1023.376,-113.514,410.014,166.149,47.970,158.672
C08527=1023.381,-113.264,410.005,166.152,47.967,158.672
C08528=1023.386,-113.015,409.997,166.155,47.963,158.672
C08529=1023.392,-112.764,409.988,166.157,47.960,158.671
C08530=1023.397,-112.515,409.980,166.160,47.957,158.671
C08531=1023.403,-112.265,409.971,166.163,47.953,158.671
C08532=1023.409,-112.015,409.962,166.166,47.950,158.671
C08533=1023.414,-111.765,409.953,166.169,47.946,158.671
C08534=1023.419,-111.516,409.945,166.173,47.943,158.671
C08535=1023.425,-111.265,409.936,166.176,47.939,158.670
C08536=1023.431,-111.016,409.927,166.179,47.936,158.670
C08537=1023.436,-110.766,409.918,166.182,47.933,158.670
C08538=1023.442,-110.516,409.909,166.185,47.930,158.670
C08539=1023.448,-110.267,409.901,166.188,47.926,158.670
C08540=1023.453,-110.018,409.892,166.191,47.923,158.670
C08541=1023.459,-109.767,409.883,166.195,47.919,158.670
C08542=1023.465,-109.517,409.875,166.197,47.916,158.669
C08543=1023.470,-109.268,409.866,166.201,47.912,158.669
C08544=1023.476,-109.018,409.857,166.203,47.910,158.669
C08545=1023.481,-108.768,409.848,166.206,47.906,158.669
C08546=1023.487,-108.518,409.840,166.209,47.902,158.669
C08547=1023.493,-108.269,409.830,166.212,47.899,158.669
C08548=1023.498,-108.019,409.822,166.215,47.895,158.668
C08549=1023.504,-107.769,409.813,166.218,47.892,158.668
C08550=1023.509,-107.519,409.804,166.221,47.889,158.668
C08551=1023.515,-107.270,409.795,166.225,47.886,158.668
C08552=1023.521,-107.019,409.786,166.228,47.882,158.668
C08553=1023.526,-106.770,409.777,166.231,47.879,158.668
C08554=1023.532,-106.520,409.768,166.234,47.876,158.667
C08555=1023.538,-106.271,409.759,166.237,47.872,158.667
C08556=1023.543,-106.020,409.750,166.240,47.869,158.667
C08557=1023.548,-105.771,409.740,166.242,47.866,158.667
C08558=1023.554,-105.521,409.732,166.246,47.862,158.667
C08559=1023.559,-105.271,409.723,166.249,47.859,158.667
C08560=1023.565,-105.022,409.714,166.252,47.855,158.666
C08561=1023.571,-104.771,409.705,166.255,47.852,158.666
C08562=1023.576,-104.522,409.696,166.258,47.849,158.666
C08563=1023.582,-104.272,409.687,166.261,47.846,158.666
C08564=1023.588,-104.023,409.678,166.264,47.842,158.666
C08565=1023.593,-103.772,409.668,166.267,47.839,158.666
C08566=1023.599,-103.523,409.659,166.271,47.836,158.666
C08567=1023.605,-103.273,409.650,166.273,47.833,158.665
C08568=1023.610,-103.023,409.641,166.276,47.830,158.665
C08569=1023.616,-102.773,409.631,166.279,47.826,158.665
C08570=1023.621,-102.524,409.623,166.282,47.823,158.665
C08571=1023.628,-102.274,409.613,166.285,47.819,158.665
C08572=1023.632,-102.024,409.604,166.289,47.816,158.665
C08573=1023.638,-101.774,409.595,166.292,47.812,158.664
C08574=1023.645,-101.489,409.585,166.295,47.809,158.664
C08575=1023.652,-101.203,409.574,166.299,47.805,158.664
C08576=1023.658,-100.917,409.563,166.302,47.801,158.664
C08577=1023.665,-100.632,409.553,166.306,47.798,158.664
C08578=1023.669,-100.382,409.543,166.309,47.794,158.663
C08579=1023.676,-100.133,409.534,166.312,47.791,158.663
C08580=1023.681,-99.883,409.525,166.314,47.788,158.663
C08581=1023.687,-99.633,409.516,166.317,47.785,158.663
C08582=1023.693,-99.383,409.506,166.320,47.781,158.663
C08583=1023.699,-99.134,409.497,166.324,47.778,158.663
C08584=1023.704,-98.883,409.488,166.327,47.774,158.663
C08585=1023.709,-98.634,409.478,166.330,47.771,158.662
C08586=1023.716,-98.385,409.469,166.333,47.767,158.662
C08587=1023.721,-98.135,409.460,166.336,47.764,158.662
C08588=1023.727,-97.885,409.451,166.339,47.761,158.662
C08589=1023.732,-97.635,409.441,166.343,47.758,158.662
C08590=1023.738,-97.386,409.431,166.344,47.754,158.661
C08591=1023.744,-97.136,409.422,166.348,47.751,158.661
C08592=1023.749,-96.885,409.412,166.351,47.748,158.661
C08593=1023.755,-96.636,409.403,166.354,47.745,158.661
C08594=1023.760,-96.386,409.393,166.357,47.742,158.661
C08595=1023.766,-96.137,409.384,166.361,47.738,158.661
C08596=1023.771,-95.887,409.374,166.363,47.736,158.661
C08597=1023.777,-95.637,409.364,166.366,47.732,158.661
C08598=1023.782,-95.388,409.354,166.369,47.729,158.660
C08599=1023.788,-95.138,409.345,166.372,47.726,158.660
C08600=1023.794,-94.888,409.335,166.376,47.723,158.660
C08601=1023.799,-94.639,409.325,166.379,47.719,158.660
C08602=1023.805,-94.388,409.317,166.382,47.716,158.660
C08603=1023.811,-94.138,409.306,166.384,47.713,158.660
C08604=1023.816,-93.889,409.297,166.387,47.710,158.659
C08605=1023.822,-93.639,409.287,166.390,47.707,158.659
C08606=1023.828,-93.389,409.277,166.394,47.703,158.659
C08607=1023.833,-93.140,409.268,166.397,47.700,158.659
C08608=1023.839,-92.890,409.258,166.400,47.697,158.659
C08609=1023.844,-92.640,409.248,166.402,47.694,158.659
C08610=1023.851,-92.390,409.238,166.405,47.690,158.659
C08611=1023.855,-92.141,409.229,166.408,47.687,158.658
C08612=1023.862,-91.891,409.219,166.412,47.684,158.658
C08613=1023.867,-91.641,409.209,166.415,47.681,158.658
C08614=1023.873,-91.392,409.200,166.418,47.678,158.658
C08615=1023.879,-91.142,409.190,166.421,47.675,158.658
C08616=1023.884,-90.892,409.179,166.423,47.672,158.658
C08617=1023.891,-90.643,409.170,166.427,47.669,158.658
C08618=1023.896,-90.393,409.160,166.430,47.665,158.657
C08619=1023.902,-90.143,409.150,166.433,47.662,158.657
C08620=1023.907,-89.893,409.140,166.436,47.658,158.657
C08621=1023.913,-89.643,409.131,166.439,47.655,158.657
C08622=1023.919,-89.393,409.120,166.441,47.652,158.657
C08623=1023.924,-89.144,409.111,166.445,47.649,158.657
C08624=1023.930,-88.894,409.101,166.448,47.646,158.656
C08625=1023.936,-88.644,409.091,166.451,47.642,158.656
C08626=1023.942,-88.395,409.081,166.454,47.639,158.656
C08627=1023.948,-88.145,409.071,166.457,47.636,158.656
C08628=1023.953,-87.896,409.061,166.461,47.633,158.656
C08629=1023.959,-87.646,409.052,166.463,47.630,158.656
C08630=1023.964,-87.396,409.041,166.466,47.627,158.656
C08631=1023.970,-87.146,409.032,166.469,47.623,158.655
C08632=1023.976,-86.896,409.021,166.472,47.620,158.655
C08633=1023.982,-86.647,409.011,166.475,47.617,158.655
C08634=1023.988,-86.397,409.001,166.479,47.613,158.655
C08635=1023.993,-86.147,408.992,166.482,47.610,158.655
C08636=1023.999,-85.897,408.982,166.485,47.606,158.654
C08637=1024.005,-85.648,408.972,166.487,47.604,158.654
C08638=1024.011,-85.364,408.960,166.491,47.600,158.654
C08639=1024.018,-85.081,408.949,166.494,47.596,158.654
C08640=1024.025,-84.798,408.937,166.498,47.592,158.654
C08641=1024.032,-84.514,408.926,166.501,47.589,158.654
C08642=1024.037,-84.265,408.917,166.504,47.586,158.653
C08643=1024.043,-84.014,408.907,166.507,47.582,158.653
C08644=1024.049,-83.765,408.896,166.511,47.579,158.653
C08645=1024.054,-83.515,408.886,166.513,47.576,158.653
C08646=1024.061,-83.265,408.877,166.516,47.573,158.653
C08647=1024.066,-83.016,408.866,166.519,47.569,158.652
C08648=1024.073,-82.766,408.856,166.522,47.566,158.652
C08649=1024.078,-82.516,408.846,166.525,47.563,158.652
C08650=1024.084,-82.267,408.836,166.529,47.560,158.652
C08651=1024.090,-82.017,408.825,166.532,47.556,158.652
C08652=1024.096,-81.767,408.816,166.534,47.553,158.652
C08653=1024.102,-81.517,408.805,166.537,47.550,158.651
C08654=1024.107,-81.267,408.795,166.540,47.547,158.651
C08655=1024.113,-81.018,408.785,166.543,47.543,158.651
C08656=1024.119,-80.768,408.774,166.546,47.540,158.651
C08657=1024.125,-80.518,408.765,166.550,47.536,158.651
C08658=1024.131,-80.269,408.754,166.553,47.533,158.651
C08659=1024.137,-80.019,408.744,166.556,47.530,158.651
C08660=1024.143,-79.769,408.734,166.558,47.527,158.650
C08661=1024.148,-79.519,408.723,166.561,47.524,158.650
C08662=1024.154,-79.270,408.712,166.565,47.521,158.650
C08663=1024.160,-79.020,408.703,166.568,47.518,158.650
C08664=1024.166,-78.771,408.692,166.571,47.515,158.650
C08665=1024.171,-78.520,408.682,166.573,47.511,158.649
C08666=1024.177,-78.271,408.671,166.576,47.508,158.649
C08667=1024.183,-78.021,408.661,166.579,47.505,158.649
C08668=1024.189,-77.772,408.651,166.583,47.502,158.649
C08669=1024.195,-77.522,408.640,166.586,47.499,158.649
C08670=1024.200,-77.272,408.630,166.588,47.496,158.649
C08671=1024.206,-77.023,408.619,166.591,47.493,158.649
C08672=1024.211,-76.772,408.608,166.595,47.490,158.648
C08673=1024.218,-76.523,408.598,166.598,47.486,158.648
C08674=1024.224,-76.274,408.587,166.601,47.483,158.648
C08675=1024.229,-76.024,408.577,166.603,47.480,158.648
C08676=1024.235,-75.774,408.566,166.606,47.477,158.648
C08677=1024.241,-75.524,408.555,166.609,47.473,158.648
C08678=1024.247,-75.274,408.545,166.613,47.470,158.647
C08679=1024.253,-75.025,408.535,166.616,47.467,158.647
C08680=1024.259,-74.775,408.524,166.618,47.464,158.647
C08681=1024.264,-74.525,408.514,166.621,47.461,158.647
C08682=1024.270,-74.276,408.503,166.625,47.458,158.647
C08683=1024.276,-74.026,408.492,166.628,47.455,158.647
C08684=1024.281,-73.776,408.482,166.630,47.452,158.646
C08685=1024.288,-73.526,408.470,166.633,47.449,158.646
C08686=1024.293,-73.276,408.460,166.636,47.446,158.646
C08687=1024.299,-73.027,408.449,166.640,47.443,158.646
C08688=1024.305,-72.777,408.438,166.642,47.440,158.646
C08689=1024.310,-72.528,408.427,166.645,47.437,158.646
C08690=1024.315,-72.277,408.416,166.649,47.434,158.646
C08691=1024.321,-72.028,408.405,166.651,47.431,158.646
C08692=1024.327,-71.779,408.394,166.654,47.428,158.645
C08693=1024.333,-71.528,408.383,166.657,47.425,158.645
C08694=1024.339,-71.279,408.372,166.660,47.422,158.645
C08695=1024.344,-71.029,408.361,166.663,47.419,158.645
C08696=1024.350,-70.780,408.350,166.666,47.416,158.645
C08697=1024.356,-70.530,408.340,166.669,47.413,158.645
C08698=1024.362,-70.281,408.329,166.671,47.410,158.644
C08699=1024.368,-70.031,408.317,166.675,47.407,158.644
C08700=1024.373,-69.781,408.306,166.678,47.404,158.644
C08701=1024.379,-69.531,408.295,166.681,47.401,158.644
C08702=1024.386,-69.250,408.283,166.684,47.397,158.644
C08703=1024.392,-68.969,408.271,166.688,47.394,158.644
C08704=1024.398,-68.687,408.258,166.690,47.390,158.644
C08705=1024.405,-68.406,408.246,166.694,47.387,158.643
C08706=1024.411,-68.156,408.235,166.697,47.384,158.643
C08707=1024.417,-67.907,408.224,166.700,47.381,158.643
C08708=1024.422,-67.657,408.213,166.702,47.378,158.643
C08709=1024.427,-67.408,408.202,166.706,47.375,158.643
C08710=1024.434,-67.157,408.191,166.709,47.372,158.643
C08711=1024.440,-66.908,408.180,166.712,47.369,158.643
C08712=1024.445,-66.658,408.169,166.714,47.366,158.642
C08713=1024.451,-66.409,408.158,166.717,47.363,158.642
C08714=1024.457,-66.159,408.147,166.721,47.360,158.642
C08715=1024.463,-65.909,408.136,166.724,47.357,158.642
C08716=1024.468,-65.659,408.124,166.726,47.354,158.642
C08717=1024.474,-65.409,408.113,166.729,47.351,158.642
C08718=1024.481,-65.160,408.102,166.733,47.348,158.641
C08719=1024.486,-64.911,408.091,166.735,47.345,158.641
C08720=1024.492,-64.661,408.080,166.738,47.342,158.641
C08721=1024.498,-64.411,408.069,166.741,47.338,158.641
C08722=1024.504,-64.162,408.058,166.744,47.335,158.641
C08723=1024.509,-63.912,408.046,166.747,47.332,158.641
C08724=1024.515,-63.662,408.035,166.750,47.329,158.640
C08725=1024.521,-63.412,408.024,166.753,47.326,158.640
C08726=1024.527,-63.163,408.013,166.756,47.323,158.640
C08727=1024.534,-62.913,408.001,166.759,47.320,158.640
C08728=1024.539,-62.664,407.990,166.762,47.317,158.640
C08729=1024.545,-62.414,407.980,166.765,47.314,158.640
C08730=1024.551,-62.164,407.968,166.767,47.311,158.639
C08731=1024.556,-61.914,407.957,166.770,47.308,158.639
C08732=1024.563,-61.665,407.945,166.774,47.305,158.639
C08733=1024.569,-61.415,407.934,166.777,47.302,158.639
C08734=1024.574,-61.166,407.923,166.779,47.299,158.639
C08735=1024.581,-60.915,407.912,166.782,47.296,158.639
C08736=1024.586,-60.666,407.900,166.786,47.293,158.639
C08737=1024.592,-60.417,407.889,166.789,47.290,158.638
C08738=1024.598,-60.167,407.878,166.791,47.287,158.638
C08739=1024.604,-59.917,407.867,166.794,47.284,158.638
C08740=1024.611,-59.668,407.855,166.798,47.281,158.638
C08741=1024.616,-59.418,407.844,166.801,47.277,158.638
C08742=1024.622,-59.168,407.832,166.803,47.275,158.638
C08743=1024.628,-58.919,407.820,166.806,47.271,158.637
C08744=1024.634,-58.669,407.810,166.809,47.268,158.637
C08745=1024.640,-58.419,407.798,166.811,47.265,158.637
C08746=1024.646,-58.169,407.787,166.815,47.262,158.637
C08747=1024.652,-57.920,407.775,166.818,47.259,158.637
C08748=1024.657,-57.670,407.764,166.821,47.256,158.636
C08749=1024.664,-57.420,407.753,166.823,47.253,158.636
C08750=1024.670,-57.171,407.741,166.827,47.250,158.636
C08751=1024.676,-56.921,407.730,166.830,47.246,158.636
C08752=1024.682,-56.672,407.718,166.833,47.243,158.636
C08753=1024.688,-56.421,407.707,166.835,47.240,158.636
C08754=1024.694,-56.172,407.696,166.838,47.237,158.635
C08755=1024.700,-55.922,407.684,166.841,47.234,158.635
C08756=1024.706,-55.673,407.673,166.845,47.230,158.635
C08757=1024.712,-55.423,407.662,166.847,47.228,158.635
C08758=1024.718,-55.174,407.650,166.850,47.225,158.635
C08759=1024.724,-54.923,407.638,166.853,47.221,158.634
C08760=1024.730,-54.674,407.627,166.857,47.218,158.634
C08761=1024.736,-54.424,407.615,166.859,47.215,158.634
C08762=1024.742,-54.175,407.604,166.862,47.212,158.634
C08763=1024.749,-53.925,407.592,166.865,47.209,158.634
C08764=1024.755,-53.675,407.580,166.868,47.205,158.634
C08765=1024.760,-53.426,407.569,166.870,47.203,158.633
C08766=1024.767,-53.146,407.556,166.874,47.199,158.633
C08767=1024.774,-52.865,407.543,166.878,47.195,158.633
C08768=1024.781,-52.585,407.530,166.881,47.192,158.633
C08769=1024.788,-52.305,407.518,166.884,47.189,158.633
C08770=1024.794,-52.055,407.505,166.887,47.185,158.632
C08771=1024.800,-51.806,407.494,166.890,47.182,158.632
C08772=1024.806,-51.556,407.482,166.892,47.179,158.632
C08773=1024.812,-51.307,407.471,166.895,47.176,158.632
C08774=1024.819,-51.057,407.459,166.899,47.173,158.632
C08775=1024.825,-50.807,407.447,166.901,47.170,158.631
C08776=1024.830,-50.558,407.436,166.904,47.167,158.631
C08777=1024.836,-50.308,407.423,166.907,47.164,158.631
C08778=1024.843,-50.058,407.412,166.909,47.161,158.631
C08779=1024.848,-49.809,407.400,166.913,47.158,158.631
C08780=1024.854,-49.559,407.387,166.916,47.155,158.631
C08781=1024.860,-49.310,407.376,166.918,47.152,158.630
C08782=1024.866,-49.026,407.362,166.921,47.149,158.630
C08783=1024.873,-48.743,407.349,166.925,47.145,158.630
C08784=1024.880,-48.460,407.335,166.929,47.142,158.630
C08785=1024.887,-48.176,407.322,166.932,47.138,158.630
C08786=1024.892,-47.927,407.309,166.934,47.135,158.629
C08787=1024.898,-47.677,407.297,166.938,47.133,158.629
C08788=1024.905,-47.428,407.285,166.941,47.130,158.629
C08789=1024.910,-47.178,407.273,166.943,47.127,158.629
C08790=1024.917,-46.928,407.261,166.946,47.124,158.629
C08791=1024.922,-46.679,407.249,166.949,47.121,158.629
C08792=1024.928,-46.429,407.237,166.952,47.118,158.629
C08793=1024.934,-46.180,407.225,166.955,47.115,158.628
C08794=1024.940,-45.930,407.212,166.957,47.112,158.628
C08795=1024.946,-45.680,407.201,166.960,47.109,158.628
C08796=1024.952,-45.430,407.189,166.964,47.106,158.628
C08797=1024.958,-45.181,407.176,166.966,47.103,158.628
C08798=1024.964,-44.932,407.165,166.969,47.100,158.627
C08799=1024.970,-44.682,407.152,166.971,47.097,158.627
C08800=1024.976,-44.432,407.140,166.975,47.094,158.627
C08801=1024.982,-44.183,407.128,166.978,47.091,158.627
C08802=1024.988,-43.933,407.115,166.980,47.088,158.627
C08803=1024.994,-43.684,407.103,166.983,47.085,158.627
C08804=1025.000,-43.433,407.092,166.987,47.082,158.626
C08805=1025.005,-43.184,407.079,166.989,47.079,158.626
C08806=1025.012,-42.934,407.067,166.992,47.076,158.626
C08807=1025.018,-42.684,407.055,166.994,47.073,158.626
C08808=1025.024,-42.435,407.043,166.997,47.070,158.626
C08809=1025.030,-42.186,407.031,167.001,47.067,158.626
C08810=1025.036,-41.936,407.018,167.003,47.064,158.625
C08811=1025.042,-41.686,407.006,167.006,47.061,158.625
C08812=1025.048,-41.436,406.994,167.009,47.058,158.625
C08813=1025.054,-41.186,406.981,167.012,47.055,158.625
C08814=1025.060,-40.938,406.970,167.015,47.052,158.625
C08815=1025.066,-40.688,406.957,167.018,47.049,158.624
C08816=1025.073,-40.438,406.945,167.020,47.046,158.624
C08817=1025.079,-40.188,406.932,167.024,47.043,158.624
C08818=1025.085,-39.938,406.920,167.026,47.040,158.624
C08819=1025.091,-39.689,406.908,167.029,47.037,158.624
C08820=1025.097,-39.440,406.896,167.032,47.034,158.624
C08821=1025.102,-39.190,406.883,167.034,47.031,158.623
C08822=1025.109,-38.940,406.871,167.038,47.028,158.623
C08823=1025.115,-38.691,406.858,167.040,47.025,158.623
C08824=1025.121,-38.441,406.845,167.043,47.022,158.623
C08825=1025.127,-38.192,406.833,167.047,47.020,158.623
C08826=1025.132,-37.943,406.820,167.049,47.017,158.623
C08827=1025.138,-37.695,406.808,167.052,47.014,158.622
C08828=1025.144,-37.448,406.796,167.054,47.011,158.622
C08829=1025.150,-37.200,406.782,167.058,47.008,158.622
C08830=1025.156,-36.952,406.771,167.060,47.005,158.622
C08831=1025.162,-36.704,406.758,167.063,47.002,158.622
C08832=1025.167,-36.456,406.746,167.066,47.000,158.622
C08833=1025.174,-36.208,406.733,167.069,46.997,158.621
C08834=1025.180,-35.959,406.720,167.071,46.994,158.621
C08835=1025.186,-35.709,406.708,167.074,46.991,158.621
C08836=1025.192,-35.459,406.695,167.076,46.988,158.621
C08837=1025.199,-35.210,406.682,167.080,46.985,158.621
C08838=1025.204,-34.961,406.670,167.083,46.982,158.621
C08839=1025.210,-34.711,406.658,167.085,46.979,158.620
C08840=1025.216,-34.461,406.645,167.088,46.976,158.620
C08841=1025.222,-34.212,406.632,167.091,46.973,158.620
C08842=1025.228,-33.962,406.619,167.094,46.971,158.620
C08843=1025.234,-33.712,406.607,167.096,46.968,158.620
C08844=1025.240,-33.463,406.593,167.100,46.965,158.620
C08845=1025.246,-33.213,406.581,167.102,46.962,158.619
C08846=1025.252,-32.963,406.568,167.105,46.959,158.619
C08847=1025.258,-32.714,406.555,167.108,46.956,158.619
C08848=1025.265,-32.464,406.543,167.111,46.953,158.619
C08849=1025.271,-32.214,406.530,167.114,46.950,158.619
C08850=1025.277,-31.965,406.517,167.116,46.947,158.618
C08851=1025.282,-31.716,406.505,167.119,46.944,158.618
C08852=1025.288,-31.466,406.492,167.121,46.942,158.618
C08853=1025.294,-31.216,406.479,167.125,46.938,158.618
C08854=1025.300,-30.967,406.467,167.128,46.935,158.618
C08855=1025.306,-30.717,406.453,167.130,46.933,158.617
C08856=1025.312,-30.467,406.441,167.133,46.929,158.617
C08857=1025.318,-30.218,406.428,167.136,46.927,158.617
C08858=1025.324,-29.968,406.415,167.139,46.924,158.617
C08859=1025.330,-29.718,406.402,167.141,46.921,158.617
C08860=1025.336,-29.469,406.389,167.144,46.918,158.617
C08861=1025.342,-29.219,406.377,167.147,46.915,158.616
C08862=1025.349,-28.970,406.364,167.150,46.912,158.616
C08863=1025.355,-28.720,406.351,167.153,46.909,158.616
C08864=1025.361,-28.471,406.338,167.155,46.906,158.616
C08865=1025.368,-28.221,406.325,167.159,46.903,158.616
C08866=1025.374,-27.971,406.312,167.161,46.900,158.615
C08867=1025.380,-27.721,406.299,167.164,46.897,158.615
C08868=1025.386,-27.472,406.286,167.166,46.894,158.615
C08869=1025.392,-27.222,406.274,167.169,46.891,158.615
C08870=1025.398,-26.973,406.260,167.172,46.889,158.615
C08871=1025.404,-26.723,406.247,167.175,46.886,158.615
C08872=1025.410,-26.474,406.234,167.177,46.883,158.614
C08873=1025.416,-26.224,406.221,167.181,46.880,158.614
C08874=1025.422,-25.974,406.208,167.183,46.877,158.614
C08875=1025.428,-25.725,406.195,167.186,46.874,158.614
C08876=1025.434,-25.476,406.181,167.188,46.871,158.614
C08877=1025.440,-25.226,406.168,167.192,46.869,158.614
C08878=1025.446,-24.976,406.155,167.194,46.866,158.613
C08879=1025.452,-24.727,406.142,167.197,46.863,158.613
C08880=1025.458,-24.477,406.129,167.200,46.860,158.613
C08881=1025.463,-24.228,406.115,167.203,46.857,158.613
C08882=1025.470,-23.978,406.102,167.205,46.854,158.613
C08883=1025.476,-23.728,406.089,167.208,46.851,158.612
C08884=1025.482,-23.479,406.076,167.211,46.849,158.612
C08885=1025.488,-23.229,406.062,167.214,46.846,158.612
C08886=1025.494,-22.980,406.049,167.216,46.843,158.612
C08887=1025.500,-22.730,406.036,167.220,46.840,158.612
C08888=1025.506,-22.481,406.023,167.222,46.837,158.611
C08889=1025.512,-22.231,406.010,167.225,46.834,158.611
C08890=1025.518,-21.982,405.996,167.227,46.832,158.611
C08891=1025.524,-21.731,405.983,167.230,46.828,158.611
C08892=1025.531,-21.482,405.970,167.233,46.826,158.611
C08893=1025.537,-21.233,405.956,167.236,46.823,158.611
C08894=1025.543,-20.952,405.941,167.238,46.820,158.610
C08895=1025.550,-20.672,405.927,167.241,46.817,158.610
C08896=1025.557,-20.390,405.911,167.245,46.814,158.610
C08897=1025.564,-20.110,405.896,167.248,46.810,158.610
C08898=1025.570,-19.861,405.883,167.251,46.807,158.610
C08899=1025.575,-19.611,405.870,167.253,46.804,158.609
C08900=1025.582,-19.361,405.856,167.256,46.801,158.609
C08901=1025.588,-19.112,405.843,167.259,46.798,158.609
C08902=1025.594,-18.862,405.830,167.262,46.796,158.609
C08903=1025.600,-18.613,405.816,167.264,46.793,158.609
C08904=1025.606,-18.364,405.803,167.268,46.790,158.608
C08905=1025.613,-18.114,405.789,167.270,46.787,158.608
C08906=1025.619,-17.864,405.776,167.273,46.784,158.608
C08907=1025.625,-17.614,405.763,167.275,46.781,158.608
C08908=1025.631,-17.365,405.749,167.279,46.778,158.608
C08909=1025.637,-17.115,405.736,167.281,46.775,158.607
C08910=1025.644,-16.866,405.723,167.284,46.772,158.607
C08911=1025.650,-16.616,405.709,167.286,46.770,158.607
C08912=1025.655,-16.367,405.695,167.289,46.766,158.607
C08913=1025.662,-16.117,405.682,167.292,46.764,158.607
C08914=1025.668,-15.868,405.668,167.295,46.761,158.606
C08915=1025.674,-15.618,405.655,167.297,46.758,158.606
C08916=1025.680,-15.369,405.641,167.299,46.755,158.606
C08917=1025.686,-15.118,405.627,167.303,46.752,158.606
C08918=1025.692,-14.869,405.614,167.305,46.749,158.606
C08919=1025.698,-14.620,405.600,167.308,46.747,158.606
C08920=1025.704,-14.370,405.587,167.311,46.744,158.605
C08921=1025.710,-14.120,405.572,167.313,46.741,158.605
C08922=1025.716,-13.871,405.559,167.316,46.738,158.605
C08923=1025.722,-13.621,405.545,167.318,46.735,158.605
C08924=1025.729,-13.371,405.532,167.322,46.732,158.605
C08925=1025.734,-13.122,405.517,167.324,46.730,158.604
C08926=1025.741,-12.873,405.504,167.327,46.727,158.604
C08927=1025.746,-12.624,405.490,167.330,46.724,158.604
C08928=1025.753,-12.374,405.476,167.332,46.722,158.604
C08929=1025.758,-12.124,405.462,167.335,46.718,158.604
C08930=1025.765,-11.875,405.449,167.337,46.716,158.603
C08931=1025.771,-11.624,405.435,167.341,46.713,158.603
C08932=1025.777,-11.376,405.421,167.343,46.710,158.603
C08933=1025.783,-11.126,405.407,167.345,46.708,158.603
C08934=1025.789,-10.876,405.393,167.349,46.705,158.603
C08935=1025.795,-10.627,405.380,167.351,46.702,158.602
C08936=1025.801,-10.377,405.366,167.354,46.699,158.602
C08937=1025.807,-10.128,405.351,167.356,46.696,158.602
C08938=1025.814,-9.878,405.338,167.360,46.693,158.602
C08939=1025.819,-9.629,405.324,167.362,46.690,158.602
C08940=1025.826,-9.379,405.311,167.364,46.687,158.601
C08941=1025.831,-9.129,405.297,167.367,46.684,158.601
C08942=1025.837,-8.880,405.282,167.369,46.682,158.601
C08943=1025.844,-8.630,405.269,167.373,46.679,158.601
C08944=1025.850,-8.381,405.255,167.375,46.676,158.601
C08945=1025.856,-8.131,405.241,167.378,46.673,158.601
C08946=1025.862,-7.882,405.226,167.381,46.671,158.600
C08947=1025.868,-7.633,405.213,167.383,46.668,158.600
C08948=1025.874,-7.382,405.199,167.386,46.665,158.600
C08949=1025.881,-7.134,405.185,167.388,46.662,158.600
C08950=1025.887,-6.883,405.171,167.392,46.659,158.600
C08951=1025.893,-6.634,405.158,167.394,46.656,158.599
C08952=1025.899,-6.385,405.144,167.396,46.653,158.599
C08953=1025.906,-6.135,405.129,167.399,46.650,158.599
C08954=1025.911,-5.886,405.115,167.402,46.647,158.599
C08955=1025.917,-5.635,405.101,167.405,46.644,158.598
C08956=1025.924,-5.387,405.087,167.407,46.642,158.598
C08957=1025.930,-5.137,405.073,167.410,46.639,158.598
C08958=1025.937,-4.855,405.058,167.413,46.636,158.598
C08959=1025.944,-4.573,405.042,167.416,46.633,158.598
C08960=1025.951,-4.290,405.026,167.419,46.629,158.597
C08961=1025.958,-4.008,405.010,167.422,46.626,158.597
C08962=1025.964,-3.758,404.996,167.424,46.623,158.597
C08963=1025.970,-3.509,404.981,167.428,46.620,158.597
C08964=1025.976,-3.259,404.967,167.430,46.618,158.597
C08965=1025.982,-3.010,404.952,167.432,46.615,158.596
C08966=1025.988,-2.760,404.938,167.436,46.612,158.596
C08967=1025.994,-2.511,404.923,167.438,46.609,158.596
C08968=1026.001,-2.261,404.910,167.440,46.607,158.596
C08969=1026.006,-2.012,404.895,167.444,46.604,158.596
C08970=1026.012,-1.762,404.881,167.446,46.601,158.596
C08971=1026.018,-1.513,404.866,167.448,46.599,158.595
C08972=1026.024,-1.264,404.852,167.451,46.596,158.595
C08973=1026.030,-1.013,404.837,167.454,46.593,158.595
C08974=1026.036,-0.764,404.823,167.456,46.591,158.595
C08975=1026.042,-0.514,404.809,167.459,46.588,158.595
C08976=1026.048,-0.265,404.794,167.462,46.585,158.594
C08977=1026.055,-0.016,404.780,167.464,46.582,158.594
C08978=1026.060,0.234,404.766,167.467,46.579,158.594
C08979=1026.067,0.483,404.751,167.470,46.577,158.594
C08980=1026.072,0.733,404.737,167.472,46.574,158.594
C08981=1026.079,0.983,404.722,167.475,46.571,158.593
C08982=1026.084,1.232,404.708,167.477,46.568,158.593
C08983=1026.090,1.482,404.693,167.479,46.566,158.593
C08984=1026.096,1.731,404.679,167.483,46.563,158.593
C08985=1026.103,1.981,404.664,167.485,46.560,158.593
C08986=1026.109,2.231,404.650,167.487,46.558,158.592
C08987=1026.114,2.480,404.635,167.491,46.555,158.592
C08988=1026.122,2.729,404.621,167.493,46.552,158.592
C08989=1026.127,2.979,404.607,167.495,46.549,158.592
C08990=1026.133,3.228,404.592,167.498,46.546,158.592
C08991=1026.139,3.477,404.577,167.501,46.544,158.592
C08992=1026.146,3.727,404.562,167.503,46.541,158.591
C08993=1026.151,3.977,404.548,167.506,46.538,158.591
C08994=1026.157,4.226,404.533,167.509,46.535,158.591
C08995=1026.164,4.476,404.519,167.511,46.533,158.591
C08996=1026.170,4.725,404.504,167.514,46.530,158.590
C08997=1026.176,4.975,404.490,167.516,46.527,158.590
C08998=1026.181,5.224,404.475,167.519,46.524,158.590
C08999=1026.188,5.474,404.460,167.522,46.521,158.590
C09000=1026.194,5.723,404.445,167.524,46.519,158.590
C09001=1026.200,5.973,404.432,167.527,46.516,158.589
C09002=1026.207,6.222,404.417,167.530,46.513,158.589
C09003=1026.213,6.471,404.402,167.532,46.510,158.589
C09004=1026.219,6.721,404.388,167.534,46.507,158.589
C09005=1026.225,6.971,404.373,167.538,46.504,158.589
C09006=1026.231,7.219,404.358,167.540,46.502,158.588
C09007=1026.237,7.470,404.344,167.542,46.499,158.588
C09008=1026.244,7.719,404.329,167.545,46.496,158.588
C09009=1026.249,7.968,404.314,167.548,46.493,158.588
C09010=1026.256,8.218,404.299,167.550,46.490,158.587
C09011=1026.262,8.468,404.284,167.553,46.487,158.587
C09012=1026.268,8.717,404.270,167.555,46.485,158.587
C09013=1026.274,8.967,404.256,167.559,46.482,158.587
C09014=1026.280,9.217,404.241,167.561,46.479,158.587
C09015=1026.286,9.466,404.226,167.563,46.477,158.586
C09016=1026.293,9.715,404.211,167.567,46.474,158.586
C09017=1026.299,9.965,404.196,167.569,46.471,158.586
C09018=1026.306,10.214,404.182,167.571,46.468,158.586
C09019=1026.312,10.463,404.167,167.574,46.465,158.586
C09020=1026.318,10.713,404.152,167.577,46.462,158.585
C09021=1026.325,10.962,404.137,167.579,46.459,158.585
C09022=1026.331,11.246,404.120,167.582,46.456,158.585
C09023=1026.339,11.530,404.104,167.585,46.453,158.585
C09024=1026.346,11.815,404.086,167.588,46.450,158.584
C09025=1026.353,12.098,404.070,167.591,46.446,158.584
C09026=1026.359,12.348,404.055,167.594,46.443,158.584
C09027=1026.365,12.598,404.040,167.596,46.440,158.584
C09028=1026.371,12.847,404.026,167.599,46.437,158.583
C09029=1026.377,13.097,404.011,167.601,46.435,158.583
C09030=1026.384,13.347,403.996,167.604,46.432,158.583
C09031=1026.390,13.596,403.981,167.607,46.429,158.583
C09032=1026.396,13.845,403.966,167.609,46.426,158.583
C09033=1026.402,14.094,403.951,167.611,46.423,158.582
C09034=1026.408,14.344,403.936,167.614,46.421,158.582
C09035=1026.415,14.594,403.921,167.617,46.418,158.582
C09036=1026.420,14.843,403.906,167.619,46.415,158.582
C09037=1026.427,15.093,403.891,167.622,46.413,158.581
C09038=1026.432,15.343,403.876,167.625,46.410,158.581
C09039=1026.439,15.592,403.861,167.627,46.407,158.581
C09040=1026.445,15.841,403.845,167.629,46.404,158.581
C09041=1026.451,16.090,403.830,167.632,46.401,158.581
C09042=1026.458,16.340,403.815,167.635,46.399,158.581
C09043=1026.463,16.590,403.800,167.637,46.396,158.580
C09044=1026.470,16.839,403.785,167.640,46.394,158.580
C09045=1026.475,17.088,403.770,167.643,46.391,158.580
C09046=1026.482,17.337,403.755,167.645,46.388,158.580
C09047=1026.488,17.587,403.739,167.647,46.385,158.579
C09048=1026.494,17.837,403.724,167.650,46.382,158.579
C09049=1026.500,18.087,403.709,167.653,46.379,158.579
C09050=1026.507,18.335,403.694,167.655,46.376,158.579
C09051=1026.512,18.585,403.678,167.657,46.374,158.578
C09052=1026.519,18.835,403.663,167.661,46.371,158.578
C09053=1026.525,19.084,403.649,167.663,46.369,158.578
C09054=1026.532,19.333,403.633,167.665,46.366,158.578
C09055=1026.537,19.583,403.617,167.668,46.363,158.578
C09056=1026.543,19.832,403.603,167.671,46.360,158.577
C09057=1026.549,20.082,403.588,167.673,46.357,158.577
C09058=1026.555,20.331,403.572,167.675,46.354,158.577
C09059=1026.562,20.581,403.557,167.678,46.352,158.577
C09060=1026.567,20.831,403.541,167.681,46.349,158.577
C09061=1026.574,21.080,403.525,167.683,46.347,158.576
C09062=1026.581,21.330,403.510,167.686,46.344,158.576
C09063=1026.586,21.578,403.495,167.688,46.341,158.576
C09064=1026.592,21.828,403.480,167.691,46.338,158.576
C09065=1026.598,22.078,403.464,167.693,46.335,158.575
C09066=1026.605,22.327,403.448,167.696,46.333,158.575
C09067=1026.611,22.577,403.433,167.698,46.330,158.575
C09068=1026.617,22.827,403.418,167.701,46.327,158.575
C09069=1026.623,23.076,403.402,167.704,46.325,158.575
C09070=1026.629,23.326,403.387,167.706,46.322,158.574
C09071=1026.635,23.574,403.371,167.708,46.319,158.574
C09072=1026.641,23.824,403.356,167.711,46.316,158.574
C09073=1026.647,24.073,403.340,167.714,46.313,158.574
C09074=1026.654,24.323,403.325,167.716,46.311,158.573
C09075=1026.659,24.573,403.310,167.718,46.308,158.573
C09076=1026.666,24.822,403.294,167.721,46.305,158.573
C09077=1026.672,25.071,403.279,167.724,46.302,158.573
C09078=1026.678,25.321,403.263,167.726,46.299,158.573
C09079=1026.685,25.570,403.248,167.729,46.296,158.572
C09080=1026.691,25.820,403.232,167.732,46.294,158.572
C09081=1026.697,26.069,403.217,167.734,46.292,158.572
C09082=1026.703,26.319,403.200,167.736,46.289,158.572
C09083=1026.709,26.568,403.186,167.739,46.286,158.572
C09084=1026.716,26.817,403.170,167.742,46.283,158.571
C09085=1026.721,27.067,403.155,167.744,46.280,158.571
C09086=1026.729,27.352,403.137,167.747,46.277,158.571
C09087=1026.736,27.637,403.119,167.749,46.274,158.570
C09088=1026.742,27.923,403.100,167.752,46.271,158.570
C09089=1026.750,28.208,403.083,167.756,46.268,158.570
C09090=1026.756,28.458,403.067,167.758,46.265,158.570
C09091=1026.761,28.707,403.051,167.760,46.262,158.570
C09092=1026.768,28.956,403.035,167.762,46.260,158.569
C09093=1026.774,29.206,403.020,167.766,46.257,158.569
C09094=1026.780,29.455,403.004,167.768,46.254,158.569
C09095=1026.786,29.705,402.988,167.770,46.252,158.569
C09096=1026.792,29.955,402.972,167.773,46.249,158.569
C09097=1026.799,30.204,402.957,167.776,46.246,158.568
C09098=1026.805,30.453,402.940,167.778,46.243,158.568
C09099=1026.810,30.703,402.925,167.780,46.240,158.568
C09100=1026.817,30.952,402.909,167.783,46.238,158.568
C09101=1026.823,31.201,402.893,167.785,46.236,158.567
C09102=1026.829,31.451,402.877,167.788,46.233,158.567
